  MoveL 4658 to (-31.93, 163.09, 78.65) mm, rotated rx 180 ry 0 rz -180 deg; joints [-126.273, -59.59, -78.383, 61.404, 66.666, -36.002]
  Call Extruder(2.36471)
  MoveL 4659 to (-32.22, 162.97, 78.65) mm, rotated rx 180 ry 0 rz 180 deg; joints [-126.252, -59.57, -78.436, 61.41, 66.694, -35.978]
  MoveL 4660 to (-32.22, 162.97, 78.65) mm, rotated rx 180 ry 0 rz 180 deg; joints [-126.252, -59.57, -78.436, 61.41, 66.694, -35.978]
  Call Extruder(2.53513)
  MoveL 4661 to (-32.49, 162.85, 78.65) mm, rotated rx -180 ry 0 rz -180 deg; joints [-126.233, -59.55, -78.486, 61.416, 66.72, -35.956]
  MoveL 4662 to (-32.49, 162.85, 78.65) mm, rotated rx -180 ry 0 rz -180 deg; joints [-126.233, -59.55, -78.486, 61.416, 66.72, -35.956]
  Call Extruder(2.69310)
  MoveL 4663 to (-32.74, 162.74, 78.65) mm, rotated rx -180 ry 0 rz 180 deg; joints [-126.215, -59.532, -78.531, 61.421, 66.744, -35.936]
  MoveL 4664 to (-32.74, 162.74, 78.65) mm, rotated rx -180 ry 0 rz 180 deg; joints [-126.215, -59.532, -78.531, 61.421, 66.744, -35.936]
  Call Extruder(2.85168)
  MoveL 4665 to (-32.99, 162.64, 78.65) mm, rotated rx 180 ry 0 rz 180 deg; joints [-126.197, -59.514, -78.577, 61.426, 66.767, -35.916]
  MoveL 4666 to (-32.99, 162.64, 78.65) mm, rotated rx 180 ry 0 rz 180 deg; joints [-126.197, -59.514, -78.577, 61.426, 66.767, -35.916]
  Call Extruder(3.05784)
  MoveL 4667 to (-33.29, 162.46, 78.65) mm, rotated rx 180 ry 0 rz -180 deg; joints [-126.179, -59.489, -78.64, 61.428, 66.797, -35.885]
  MoveL 4668 to (-33.29, 162.46, 78.65) mm, rotated rx 180 ry 0 rz -180 deg; joints [-126.179, -59.489, -78.64, 61.428, 66.797, -35.885]
  Call Extruder(3.26479)
  MoveL 4669 to (-33.6, 162.29, 78.65) mm, rotated rx 180 ry 0 rz -180 deg; joints [-126.16, -59.465, -78.703, 61.43, 66.826, -35.855]
  MoveL 4670 to (-33.6, 162.29, 78.65) mm, rotated rx 180 ry 0 rz -180 deg; joints [-126.16, -59.465, -78.703, 61.43, 66.826, -35.855]
  Call Extruder(3.47251)
  MoveL 4671 to (-33.9, 162.11, 78.65) mm, rotated rx 180 ry 0 rz 180 deg; joints [-126.142, -59.44, -78.766, 61.432, 66.855, -35.825]
  MoveL 4672 to (-33.9, 162.11, 78.65) mm, rotated rx 180 ry 0 rz 180 deg; joints [-126.142, -59.44, -78.766, 61.432, 66.855, -35.825]
  Call Extruder(3.68102)
  MoveL 4673 to (-34.21, 161.93, 78.65) mm, rotated rx -180 ry 0 rz 180 deg; joints [-126.123, -59.415, -78.829, 61.434, 66.884, -35.795]
  MoveL 4674 to (-34.21, 161.93, 78.65) mm, rotated rx -180 ry 0 rz 180 deg; joints [-126.123, -59.415, -78.829, 61.434, 66.884, -35.795]
  Call Extruder(3.86055)
  MoveL 4675 to (-34.45, 161.76, 78.65) mm, rotated rx -180 ry 0 rz 180 deg; joints [-126.111, -59.393, -78.885, 61.432, 66.907, -35.767]
  MoveL 4676 to (-34.45, 161.76, 78.65) mm, rotated rx -180 ry 0 rz 180 deg; joints [-126.111, -59.393, -78.885, 61.432, 66.907, -35.767]
  Call Extruder(4.19399)
  MoveL 4677 to (-34.9, 161.43, 78.65) mm, rotated rx 180 ry 0 rz 180 deg; joints [-126.089, -59.353, -78.988, 61.428, 66.95, -35.714]
  MoveL 4678 to (-34.9, 161.43, 78.65) mm, rotated rx 180 ry 0 rz 180 deg; joints [-126.089, -59.353, -78.988, 61.428, 66.95, -35.714]
  Call Extruder(4.52861)
  MoveL 4679 to (-35.35, 161.1, 78.65) mm, rotated rx 180 ry 0 rz -180 deg; joints [-126.067, -59.312, -79.092, 61.424, 66.993, -35.662]
  Call Extruder(5.35652)
  MoveL 4680 to (-36.39, 160.19, 78.65) mm, rotated rx -180 ry 0 rz 180 deg; joints [-126.027, -59.21, -79.355, 61.399, 67.093, -35.523]
  Call Extruder(6.18445)
  MoveL 4681 to (-37.3, 159.15, 78.65) mm, rotated rx -180 ry 0 rz 180 deg; joints [-126.011, -59.106, -79.622, 61.354, 67.181, -35.373]
  Call Extruder(6.35176)
  MoveL 4682 to (-37.47, 158.93, 78.65) mm, rotated rx 180 ry 0 rz 180 deg; joints [-126.011, -59.084, -79.676, 61.341, 67.197, -35.341]
  MoveL 4683 to (-37.47, 158.93, 78.65) mm, rotated rx 180 ry 0 rz 180 deg; joints [-126.011, -59.084, -79.676, 61.341, 67.197, -35.341]
  Call Extruder(6.68519)
  MoveL 4684 to (-37.79, 158.48, 78.65) mm, rotated rx 180 ry 0 rz -180 deg; joints [-126.011, -59.042, -79.784, 61.317, 67.228, -35.279]
  MoveL 4685 to (-37.79, 158.48, 78.65) mm, rotated rx 180 ry 0 rz -180 deg; joints [-126.011, -59.042, -79.784, 61.317, 67.228, -35.279]
  Call Extruder(7.01743)
  MoveL 4686 to (-38.12, 158.02, 78.65) mm, rotated rx 180 ry 0 rz -180 deg; joints [-126.011, -59, -79.893, 61.293, 67.26, -35.216]
  MoveL 4687 to (-38.12, 158.02, 78.65) mm, rotated rx 180 ry 0 rz -180 deg; joints [-126.011, -59, -79.893, 61.293, 67.26, -35.216]
  Call Extruder(7.13511)
  MoveL 4688 to (-38.22, 157.85, 78.65) mm, rotated rx 180 ry 0 rz 180 deg; joints [-126.013, -58.986, -79.931, 61.282, 67.27, -35.192]
  MoveL 4689 to (-38.22, 157.85, 78.65) mm, rotated rx 180 ry 0 rz 180 deg; joints [-126.013, -58.986, -79.931, 61.282, 67.27, -35.192]
  Call Extruder(7.34283)
  MoveL 4690 to (-38.4, 157.55, 78.65) mm, rotated rx 180 ry 0 rz -180 deg; joints [-126.018, -58.959, -79.998, 61.262, 67.287, -35.151]
  MoveL 4691 to (-38.4, 157.55, 78.65) mm, rotated rx 180 ry 0 rz -180 deg; joints [-126.018, -58.959, -79.998, 61.262, 67.287, -35.151]
  Call Extruder(7.54978)
  MoveL 4692 to (-38.57, 157.25, 78.65) mm, rotated rx 180 ry 0 rz 180 deg; joints [-126.023, -58.933, -80.066, 61.243, 67.304, -35.111]
  MoveL 4693 to (-38.57, 157.25, 78.65) mm, rotated rx 180 ry 0 rz 180 deg; joints [-126.023, -58.933, -80.066, 61.243, 67.304, -35.111]
  Call Extruder(7.75595)
  MoveL 4694 to (-38.75, 156.94, 78.65) mm, rotated rx -180 ry 0 rz 180 deg; joints [-126.028, -58.907, -80.133, 61.223, 67.321, -35.07]
  MoveL 4695 to (-38.75, 156.94, 78.65) mm, rotated rx -180 ry 0 rz 180 deg; joints [-126.028, -58.907, -80.133, 61.223, 67.321, -35.07]
  Call Extruder(7.93762)
  MoveL 4696 to (-38.89, 156.66, 78.65) mm, rotated rx 180 ry 0 rz 180 deg; joints [-126.034, -58.884, -80.193, 61.204, 67.335, -35.033]
  MoveL 4697 to (-38.89, 156.66, 78.65) mm, rotated rx 180 ry 0 rz 180 deg; joints [-126.034, -58.884, -80.193, 61.204, 67.335, -35.033]
  Call Extruder(8.09561)
  MoveL 4698 to (-39, 156.42, 78.65) mm, rotated rx 180 ry 0 rz -180 deg; joints [-126.042, -58.864, -80.244, 61.186, 67.345, -35]
  MoveL 4699 to (-39, 156.42, 78.65) mm, rotated rx 180 ry 0 rz -180 deg; joints [-126.042, -58.864, -80.244, 61.186, 67.345, -35]
  Call Extruder(8.25300)
  MoveL 4700 to (-39.1, 156.17, 78.65) mm, rotated rx 180 ry 0 rz 180 deg; joints [-126.05, -58.845, -80.295, 61.167, 67.356, -34.968]
  MoveL 4701 to (-39.1, 156.17, 78.65) mm, rotated rx 180 ry 0 rz 180 deg; joints [-126.05, -58.845, -80.295, 61.167, 67.356, -34.968]
  Call Extruder(8.43572)
  MoveL 4702 to (-39.23, 155.88, 78.65) mm, rotated rx 180 ry 0 rz 180 deg; joints [-126.06, -58.822, -80.354, 61.145, 67.368, -34.93]
  MoveL 4703 to (-39.23, 155.88, 78.65) mm, rotated rx 180 ry 0 rz 180 deg; joints [-126.06, -58.822, -80.354, 61.145, 67.368, -34.93]
  Call Extruder(8.61768)
  MoveL 4704 to (-39.35, 155.58, 78.65) mm, rotated rx -180 ry 0 rz -180 deg; joints [-126.07, -58.799, -80.413, 61.123, 67.38, -34.892]
  MoveL 4705 to (-39.35, 155.58, 78.65) mm, rotated rx -180 ry 0 rz -180 deg; joints [-126.07, -58.799, -80.413, 61.123, 67.38, -34.892]
  Call Extruder(8.76501)
  MoveL 4706 to (-39.44, 155.34, 78.65) mm, rotated rx 180 ry 0 rz 180 deg; joints [-126.079, -58.78, -80.461, 61.105, 67.389, -34.862]
  MoveL 4707 to (-39.44, 155.34, 78.65) mm, rotated rx 180 ry 0 rz 180 deg; joints [-126.079, -58.78, -80.461, 61.105, 67.389, -34.862]
  Call Extruder(8.87825)
  MoveL 4708 to (-39.5, 155.15, 78.65) mm, rotated rx -180 ry 0 rz 180 deg; joints [-126.087, -58.766, -80.497, 61.089, 67.395, -34.838]
  MoveL 4709 to (-39.5, 155.15, 78.65) mm, rotated rx -180 ry 0 rz 180 deg; joints [-126.087, -58.766, -80.497, 61.089, 67.395, -34.838]
  Call Extruder(8.99103)
  MoveL 4710 to (-39.56, 154.97, 78.65) mm, rotated rx 180 ry 0 rz 180 deg; joints [-126.095, -58.752, -80.533, 61.074, 67.401, -34.814]
  MoveL 4711 to (-39.56, 154.97, 78.65) mm, rotated rx 180 ry 0 rz 180 deg; joints [-126.095, -58.752, -80.533, 61.074, 67.401, -34.814]
  Call Extruder(9.10338)
  MoveL 4712 to (-39.62, 154.78, 78.65) mm, rotated rx 180 ry 0 rz 180 deg; joints [-126.103, -58.738, -80.57, 61.059, 67.407, -34.79]
  MoveL 4713 to (-39.62, 154.78, 78.65) mm, rotated rx 180 ry 0 rz 180 deg; joints [-126.103, -58.738, -80.57, 61.059, 67.407, -34.79]
  Call Extruder(9.21528)
  MoveL 4714 to (-39.68, 154.59, 78.65) mm, rotated rx -180 ry 0 rz 180 deg; joints [-126.111, -58.725, -80.606, 61.043, 67.413, -34.766]
  MoveL 4715 to (-39.68, 154.59, 78.65) mm, rotated rx -180 ry 0 rz 180 deg; joints [-126.111, -58.725, -80.606, 61.043, 67.413, -34.766]
  Call Extruder(9.33668)
  MoveL 4716 to (-39.75, 154.38, 78.65) mm, rotated rx -180 ry 0 rz 180 deg; joints [-126.12, -58.709, -80.645, 61.026, 67.42, -34.74]
  MoveL 4717 to (-39.75, 154.38, 78.65) mm, rotated rx -180 ry 0 rz 180 deg; joints [-126.12, -58.709, -80.645, 61.026, 67.42, -34.74]
  Call Extruder(9.46748)
  MoveL 4718 to (-39.81, 154.16, 78.65) mm, rotated rx 180 ry 0 rz 180 deg; joints [-126.131, -58.693, -80.688, 61.008, 67.427, -34.712]
  MoveL 4719 to (-39.81, 154.16, 78.65) mm, rotated rx 180 ry 0 rz 180 deg; joints [-126.131, -58.693, -80.688, 61.008, 67.427, -34.712]
  Call Extruder(9.59770)
  MoveL 4720 to (-39.88, 153.94, 78.65) mm, rotated rx 180 ry 0 rz 180 deg; joints [-126.141, -58.677, -80.73, 60.989, 67.433, -34.684]
  MoveL 4721 to (-39.88, 153.94, 78.65) mm, rotated rx 180 ry 0 rz 180 deg; joints [-126.141, -58.677, -80.73, 60.989, 67.433, -34.684]
  Call Extruder(9.72737)
  MoveL 4722 to (-39.95, 153.71, 78.65) mm, rotated rx 180 ry 0 rz 180 deg; joints [-126.151, -58.66, -80.772, 60.971, 67.44, -34.655]
  MoveL 4723 to (-39.95, 153.71, 78.65) mm, rotated rx 180 ry 0 rz 180 deg; joints [-126.151, -58.66, -80.772, 60.971, 67.44, -34.655]
  Call Extruder(9.85647)
  MoveL 4724 to (-40.02, 153.49, 78.65) mm, rotated rx -180 ry 0 rz -180 deg; joints [-126.161, -58.644, -80.815, 60.952, 67.447, -34.627]
  MoveL 4725 to (-40.02, 153.49, 78.65) mm, rotated rx -180 ry 0 rz -180 deg; joints [-126.161, -58.644, -80.815, 60.952, 67.447, -34.627]
  Call Extruder(9.97156)
  MoveL 4726 to (-40.06, 153.28, 78.65) mm, rotated rx -180 ry 0 rz 180 deg; joints [-126.173, -58.63, -80.851, 60.934, 67.452, -34.602]
  MoveL 4727 to (-40.06, 153.28, 78.65) mm, rotated rx -180 ry 0 rz 180 deg; joints [-126.173, -58.63, -80.851, 60.934, 67.452, -34.602]
  Call Extruder(10.08619)
  MoveL 4728 to (-40.11, 153.08, 78.65) mm, rotated rx 180 ry 0 rz -180 deg; joints [-126.184, -58.616, -80.888, 60.916, 67.456, -34.577]
  MoveL 4729 to (-40.11, 153.08, 78.65) mm, rotated rx 180 ry 0 rz -180 deg; joints [-126.184, -58.616, -80.888, 60.916, 67.456, -34.577]
  Call Extruder(10.20037)
  MoveL 4730 to (-40.15, 152.88, 78.65) mm, rotated rx 180 ry 0 rz 180 deg; joints [-126.195, -58.602, -80.925, 60.897, 67.461, -34.552]
  MoveL 4731 to (-40.15, 152.88, 78.65) mm, rotated rx 180 ry 0 rz 180 deg; joints [-126.195, -58.602, -80.925, 60.897, 67.461, -34.552]
  Call Extruder(10.31410)
  MoveL 4732 to (-40.2, 152.67, 78.65) mm, rotated rx 180 ry 0 rz 180 deg; joints [-126.206, -58.588, -80.961, 60.879, 67.465, -34.526]
  MoveL 4733 to (-40.2, 152.67, 78.65) mm, rotated rx 180 ry 0 rz 180 deg; joints [-126.206, -58.588, -80.961, 60.879, 67.465, -34.526]
  Call Extruder(10.43953)
  MoveL 4734 to (-40.24, 152.44, 78.65) mm, rotated rx 180 ry 0 rz 180 deg; joints [-126.219, -58.572, -81.002, 60.859, 67.47, -34.499]
  MoveL 4735 to (-40.24, 152.44, 78.65) mm, rotated rx 180 ry 0 rz 180 deg; joints [-126.219, -58.572, -81.002, 60.859, 67.47, -34.499]
  Call Extruder(10.57650)
  MoveL 4736 to (-40.29, 152.2, 78.65) mm, rotated rx 180 ry 0 rz -180 deg; joints [-126.233, -58.555, -81.046, 60.836, 67.476, -34.468]
  MoveL 4737 to (-40.29, 152.2, 78.65) mm, rotated rx 180 ry 0 rz -180 deg; joints [-126.233, -58.555, -81.046, 60.836, 67.476, -34.468]
  Call Extruder(10.71287)
  MoveL 4738 to (-40.34, 151.95, 78.65) mm, rotated rx 180 ry 0 rz 180 deg; joints [-126.248, -58.538, -81.09, 60.814, 67.481, -34.437]
  MoveL 4739 to (-40.34, 151.95, 78.65) mm, rotated rx 180 ry 0 rz 180 deg; joints [-126.248, -58.538, -81.09, 60.814, 67.481, -34.437]
  Call Extruder(10.84862)
  MoveL 4740 to (-40.39, 151.7, 78.65) mm, rotated rx 180 ry 0 rz 180 deg; joints [-126.262, -58.521, -81.134, 60.791, 67.486, -34.407]
  MoveL 4741 to (-40.39, 151.7, 78.65) mm, rotated rx 180 ry 0 rz 180 deg; joints [-126.262, -58.521, -81.134, 60.791, 67.486, -34.407]
  Call Extruder(10.98377)
  MoveL 4742 to (-40.44, 151.45, 78.65) mm, rotated rx 180 ry 0 rz 180 deg; joints [-126.276, -58.505, -81.178, 60.768, 67.491, -34.376]
  MoveL 4743 to (-40.44, 151.45, 78.65) mm, rotated rx 180 ry 0 rz 180 deg; joints [-126.276, -58.505, -81.178, 60.768, 67.491, -34.376]
  Call Extruder(11.11830)
  MoveL 4744 to (-40.49, 151.2, 78.65) mm, rotated rx 180 ry 0 rz 180 deg; joints [-126.291, -58.488, -81.222, 60.746, 67.496, -34.346]
  MoveL 4745 to (-40.49, 151.2, 78.65) mm, rotated rx 180 ry 0 rz 180 deg; joints [-126.291, -58.488, -81.222, 60.746, 67.496, -34.346]
  Call Extruder(11.25223)
  MoveL 4746 to (-40.54, 150.95, 78.65) mm, rotated rx -180 ry 0 rz 180 deg; joints [-126.305, -58.471, -81.266, 60.723, 67.501, -34.315]
  MoveL 4747 to (-40.54, 150.95, 78.65) mm, rotated rx -180 ry 0 rz 180 deg; joints [-126.305, -58.471, -81.266, 60.723, 67.501, -34.315]
  Call Extruder(11.40008)
  MoveL 4748 to (-40.59, 150.67, 78.65) mm, rotated rx -180 ry 0 rz 180 deg; joints [-126.322, -58.452, -81.314, 60.697, 67.506, -34.281]
  MoveL 4749 to (-40.59, 150.67, 78.65) mm, rotated rx -180 ry 0 rz 180 deg; joints [-126.322, -58.452, -81.314, 60.697, 67.506, -34.281]
  Call Extruder(11.56181)
  MoveL 4750 to (-40.64, 150.37, 78.65) mm, rotated rx -180 ry 0 rz -180 deg; joints [-126.341, -58.432, -81.367, 60.669, 67.512, -34.244]
  MoveL 4751 to (-40.64, 150.37, 78.65) mm, rotated rx -180 ry 0 rz -180 deg; joints [-126.341, -58.432, -81.367, 60.669, 67.512, -34.244]
  Call Extruder(11.72281)
  MoveL 4752 to (-40.69, 150.06, 78.65) mm, rotated rx 180 ry 0 rz -180 deg; joints [-126.36, -58.412, -81.419, 60.64, 67.517, -34.207]
  MoveL 4753 to (-40.69, 150.06, 78.65) mm, rotated rx 180 ry 0 rz -180 deg; joints [-126.36, -58.412, -81.419, 60.64, 67.517, -34.207]
  Call Extruder(11.88308)
  MoveL 4754 to (-40.74, 149.76, 78.65) mm, rotated rx -180 ry 0 rz 180 deg; joints [-126.379, -58.392, -81.472, 60.611, 67.522, -34.17]
  MoveL 4755 to (-40.74, 149.76, 78.65) mm, rotated rx -180 ry 0 rz 180 deg; joints [-126.379, -58.392, -81.472, 60.611, 67.522, -34.17]
  Call Extruder(12.04262)
  MoveL 4756 to (-40.78, 149.45, 78.65) mm, rotated rx 180 ry 0 rz 180 deg; joints [-126.398, -58.372, -81.524, 60.583, 67.527, -34.133]
  MoveL 4757 to (-40.78, 149.45, 78.65) mm, rotated rx 180 ry 0 rz 180 deg; joints [-126.398, -58.372, -81.524, 60.583, 67.527, -34.133]
  Call Extruder(12.20143)
  MoveL 4758 to (-40.83, 149.14, 78.65) mm, rotated rx -180 ry 0 rz 180 deg; joints [-126.417, -58.352, -81.577, 60.554, 67.533, -34.096]
  MoveL 4759 to (-40.83, 149.14, 78.65) mm, rotated rx -180 ry 0 rz 180 deg; joints [-126.417, -58.352, -81.577, 60.554, 67.533, -34.096]
  Call Extruder(12.38010)
  MoveL 4760 to (-40.88, 148.8, 78.65) mm, rotated rx -180 ry 0 rz 180 deg; joints [-126.439, -58.33, -81.635, 60.521, 67.538, -34.054]
  MoveL 4761 to (-40.88, 148.8, 78.65) mm, rotated rx -180 ry 0 rz 180 deg; joints [-126.439, -58.33, -81.635, 60.521, 67.538, -34.054]
  Call Extruder(12.57854)
  MoveL 4762 to (-40.92, 148.41, 78.65) mm, rotated rx 180 ry 0 rz -180 deg; joints [-126.465, -58.305, -81.7, 60.483, 67.543, -34.008]
  MoveL 4763 to (-40.92, 148.41, 78.65) mm, rotated rx 180 ry 0 rz -180 deg; joints [-126.465, -58.305, -81.7, 60.483, 67.543, -34.008]
  Call Extruder(12.77611)
  MoveL 4764 to (-40.97, 148.02, 78.65) mm, rotated rx 180 ry 0 rz -180 deg; joints [-126.491, -58.281, -81.764, 60.445, 67.548, -33.961]
  MoveL 4765 to (-40.97, 148.02, 78.65) mm, rotated rx 180 ry 0 rz -180 deg; joints [-126.491, -58.281, -81.764, 60.445, 67.548, -33.961]
  Call Extruder(12.97282)
  MoveL 4766 to (-41.02, 147.63, 78.65) mm, rotated rx 180 ry 0 rz 180 deg; joints [-126.517, -58.256, -81.829, 60.408, 67.553, -33.915]
  MoveL 4767 to (-41.02, 147.63, 78.65) mm, rotated rx 180 ry 0 rz 180 deg; joints [-126.517, -58.256, -81.829, 60.408, 67.553, -33.915]
  Call Extruder(13.16866)
  MoveL 4768 to (-41.06, 147.25, 78.65) mm, rotated rx -180 ry 0 rz -180 deg; joints [-126.543, -58.232, -81.893, 60.37, 67.558, -33.868]
  MoveL 4769 to (-41.06, 147.25, 78.65) mm, rotated rx -180 ry 0 rz -180 deg; joints [-126.543, -58.232, -81.893, 60.37, 67.558, -33.868]
  Call Extruder(13.46406)
  MoveL 4770 to (-41.11, 146.66, 78.65) mm, rotated rx -180 ry 0 rz -180 deg; joints [-126.585, -58.195, -81.988, 60.311, 67.564, -33.798]
  MoveL 4771 to (-41.11, 146.66, 78.65) mm, rotated rx -180 ry 0 rz -180 deg; joints [-126.585, -58.195, -81.988, 60.311, 67.564, -33.798]
  Call Extruder(13.75812)
  MoveL 4772 to (-41.15, 146.07, 78.65) mm, rotated rx -180 ry 0 rz -180 deg; joints [-126.628, -58.159, -82.083, 60.252, 67.57, -33.728]
  MoveL 4773 to (-41.15, 146.07, 78.65) mm, rotated rx -180 ry 0 rz -180 deg; joints [-126.628, -58.159, -82.083, 60.252, 67.57, -33.728]
  Call Extruder(14.05086)
  MoveL 4774 to (-41.2, 145.48, 78.65) mm, rotated rx 180 ry 0 rz 180 deg; joints [-126.67, -58.123, -82.178, 60.192, 67.576, -33.658]
  MoveL 4775 to (-41.2, 145.48, 78.65) mm, rotated rx 180 ry 0 rz 180 deg; joints [-126.67, -58.123, -82.178, 60.192, 67.576, -33.658]
  Call Extruder(14.62431)
  MoveL 4776 to (-41.25, 144.32, 78.65) mm, rotated rx 180 ry 0 rz 180 deg; joints [-126.759, -58.054, -82.36, 60.072, 67.583, -33.522]
  MoveL 4777 to (-41.25, 144.32, 78.65) mm, rotated rx 180 ry 0 rz 180 deg; joints [-126.759, -58.054, -82.36, 60.072, 67.583, -33.522]
  Call Extruder(15.33827)
  MoveL 4778 to (-41.29, 142.86, 78.65) mm, rotated rx 180 ry 0 rz -180 deg; joints [-126.873, -57.969, -82.585, 59.919, 67.59, -33.352]
  Call Extruder(57.40309)
  MoveL 4779 to (-41.29, 57.14, 78.65) mm, rotated rx 180 ry 0 rz 180 deg; joints [-135.148, -53.894, -94.222, 49.519, 68.009, -23.688]
  Call Extruder(57.83164)
  MoveL 4780 to (-41.27, 56.26, 78.65) mm, rotated rx -180 ry 0 rz -180 deg; joints [-135.25, -53.862, -94.325, 49.397, 68.014, -23.593]
  MoveL 4781 to (-41.27, 56.26, 78.65) mm, rotated rx -180 ry 0 rz -180 deg; joints [-135.25, -53.862, -94.325, 49.397, 68.014, -23.593]
  Call Extruder(58.40509)
  MoveL 4782 to (-41.22, 55.1, 78.65) mm, rotated rx 180 ry 0 rz 180 deg; joints [-135.387, -53.819, -94.459, 49.232, 68.019, -23.467]
  MoveL 4783 to (-41.22, 55.1, 78.65) mm, rotated rx 180 ry 0 rz 180 deg; joints [-135.387, -53.819, -94.459, 49.232, 68.019, -23.467]
  Call Extruder(58.83941)
  MoveL 4784 to (-41.18, 54.23, 78.65) mm, rotated rx 180 ry 0 rz 180 deg; joints [-135.493, -53.788, -94.558, 49.107, 68.021, -23.372]
  MoveL 4785 to (-41.18, 54.23, 78.65) mm, rotated rx 180 ry 0 rz 180 deg; joints [-135.493, -53.788, -94.558, 49.107, 68.021, -23.372]
  Call Extruder(59.13347)
  MoveL 4786 to (-41.13, 53.64, 78.65) mm, rotated rx -180 ry 0 rz 180 deg; joints [-135.566, -53.767, -94.623, 49.021, 68.021, -23.309]
  MoveL 4787 to (-41.13, 53.64, 78.65) mm, rotated rx -180 ry 0 rz 180 deg; joints [-135.566, -53.767, -94.623, 49.021, 68.021, -23.309]
  Call Extruder(59.42887)
  MoveL 4788 to (-41.09, 53.05, 78.65) mm, rotated rx 180 ry 0 rz 180 deg; joints [-135.64, -53.747, -94.687, 48.935, 68.021, -23.246]
  MoveL 4789 to (-41.09, 53.05, 78.65) mm, rotated rx 180 ry 0 rz 180 deg; joints [-135.64, -53.747, -94.687, 48.935, 68.021, -23.246]
  Call Extruder(59.67511)
  MoveL 4790 to (-41.04, 52.56, 78.65) mm, rotated rx 180 ry 0 rz 180 deg; joints [-135.701, -53.731, -94.74, 48.863, 68.021, -23.194]
  MoveL 4791 to (-41.04, 52.56, 78.65) mm, rotated rx 180 ry 0 rz 180 deg; joints [-135.701, -53.731, -94.74, 48.863, 68.021, -23.194]
  Call Extruder(59.87182)
  MoveL 4792 to (-40.99, 52.17, 78.65) mm, rotated rx 180 ry 0 rz 180 deg; joints [-135.751, -53.718, -94.78, 48.805, 68.019, -23.153]
  MoveL 4793 to (-40.99, 52.17, 78.65) mm, rotated rx 180 ry 0 rz 180 deg; joints [-135.751, -53.718, -94.78, 48.805, 68.019, -23.153]
  Call Extruder(60.06939)
  MoveL 4794 to (-40.95, 51.78, 78.65) mm, rotated rx -180 ry 0 rz -180 deg; joints [-135.801, -53.705, -94.82, 48.747, 68.018, -23.112]
  MoveL 4795 to (-40.95, 51.78, 78.65) mm, rotated rx -180 ry 0 rz -180 deg; joints [-135.801, -53.705, -94.82, 48.747, 68.018, -23.112]
  Call Extruder(60.26783)
  MoveL 4796 to (-40.9, 51.4, 78.65) mm, rotated rx 180 ry 0 rz -180 deg; joints [-135.852, -53.692, -94.861, 48.689, 68.016, -23.071]
  MoveL 4797 to (-40.9, 51.4, 78.65) mm, rotated rx 180 ry 0 rz -180 deg; joints [-135.852, -53.692, -94.861, 48.689, 68.016, -23.071]
  Call Extruder(60.46714)
  MoveL 4798 to (-40.86, 51.01, 78.65) mm, rotated rx -180 ry 0 rz 180 deg; joints [-135.902, -53.68, -94.901, 48.63, 68.015, -23.03]
  MoveL 4799 to (-40.86, 51.01, 78.65) mm, rotated rx -180 ry 0 rz 180 deg; joints [-135.902, -53.68, -94.901, 48.63, 68.015, -23.03]
  Call Extruder(60.62596)
  MoveL 4800 to (-40.81, 50.7, 78.65) mm, rotated rx 180 ry 0 rz -180 deg; joints [-135.943, -53.67, -94.931, 48.583, 68.012, -22.998]
  MoveL 4801 to (-40.81, 50.7, 78.65) mm, rotated rx 180 ry 0 rz -180 deg; joints [-135.943, -53.67, -94.931, 48.583, 68.012, -22.998]
  Call Extruder(60.78550)
  MoveL 4802 to (-40.76, 50.4, 78.65) mm, rotated rx 180 ry 0 rz -180 deg; joints [-135.984, -53.661, -94.961, 48.536, 68.01, -22.966]
  MoveL 4803 to (-40.76, 50.4, 78.65) mm, rotated rx 180 ry 0 rz -180 deg; joints [-135.984, -53.661, -94.961, 48.536, 68.01, -22.966]
  Call Extruder(60.94577)
  MoveL 4804 to (-40.71, 50.09, 78.65) mm, rotated rx 180 ry 0 rz 180 deg; joints [-136.025, -53.652, -94.992, 48.489, 68.008, -22.934]
  MoveL 4805 to (-40.71, 50.09, 78.65) mm, rotated rx 180 ry 0 rz 180 deg; joints [-136.025, -53.652, -94.992, 48.489, 68.008, -22.934]
  Call Extruder(61.10677)
  MoveL 4806 to (-40.66, 49.79, 78.65) mm, rotated rx 180 ry 0 rz -180 deg; joints [-136.067, -53.642, -95.022, 48.442, 68.005, -22.902]
  MoveL 4807 to (-40.66, 49.79, 78.65) mm, rotated rx 180 ry 0 rz -180 deg; joints [-136.067, -53.642, -95.022, 48.442, 68.005, -22.902]
  Call Extruder(61.26850)
  MoveL 4808 to (-40.61, 49.48, 78.65) mm, rotated rx 180 ry 0 rz 180 deg; joints [-136.108, -53.633, -95.052, 48.395, 68.003, -22.87]
  MoveL 4809 to (-40.61, 49.48, 78.65) mm, rotated rx 180 ry 0 rz 180 deg; joints [-136.108, -53.633, -95.052, 48.395, 68.003, -22.87]
  Call Extruder(61.43095)
  MoveL 4810 to (-40.56, 49.18, 78.65) mm, rotated rx 180 ry 0 rz 180 deg; joints [-136.149, -53.623, -95.082, 48.347, 68.001, -22.838]
  MoveL 4811 to (-40.56, 49.18, 78.65) mm, rotated rx 180 ry 0 rz 180 deg; joints [-136.149, -53.623, -95.082, 48.347, 68.001, -22.838]
  Call Extruder(61.56487)
  MoveL 4812 to (-40.52, 48.92, 78.65) mm, rotated rx -180 ry 0 rz 180 deg; joints [-136.184, -53.616, -95.105, 48.308, 67.998, -22.812]
  MoveL 4813 to (-40.52, 48.92, 78.65) mm, rotated rx -180 ry 0 rz 180 deg; joints [-136.184, -53.616, -95.105, 48.308, 67.998, -22.812]
  Call Extruder(61.69941)
  MoveL 4814 to (-40.47, 48.68, 78.65) mm, rotated rx -180 ry 0 rz 180 deg; joints [-136.219, -53.609, -95.128, 48.269, 67.995, -22.786]
  MoveL 4815 to (-40.47, 48.68, 78.65) mm, rotated rx -180 ry 0 rz 180 deg; joints [-136.219, -53.609, -95.128, 48.269, 67.995, -22.786]
  Call Extruder(61.83455)
  MoveL 4816 to (-40.42, 48.43, 78.65) mm, rotated rx 180 ry 0 rz 180 deg; joints [-136.254, -53.602, -95.151, 48.229, 67.992, -22.76]
  MoveL 4817 to (-40.42, 48.43, 78.65) mm, rotated rx 180 ry 0 rz 180 deg; joints [-136.254, -53.602, -95.151, 48.229, 67.992, -22.76]
  Call Extruder(61.97031)
  MoveL 4818 to (-40.37, 48.18, 78.65) mm, rotated rx 180 ry 0 rz 180 deg; joints [-136.288, -53.594, -95.174, 48.19, 67.989, -22.734]
  MoveL 4819 to (-40.37, 48.18, 78.65) mm, rotated rx 180 ry 0 rz 180 deg; joints [-136.288, -53.594, -95.174, 48.19, 67.989, -22.734]
  Call Extruder(62.10667)
  MoveL 4820 to (-40.32, 47.93, 78.65) mm, rotated rx -180 ry 0 rz 180 deg; joints [-136.323, -53.587, -95.197, 48.15, 67.986, -22.709]
  MoveL 4821 to (-40.32, 47.93, 78.65) mm, rotated rx -180 ry 0 rz 180 deg; joints [-136.323, -53.587, -95.197, 48.15, 67.986, -22.709]
  Call Extruder(62.24365)
  MoveL 4822 to (-40.27, 47.68, 78.65) mm, rotated rx 180 ry 0 rz 180 deg; joints [-136.358, -53.58, -95.221, 48.111, 67.983, -22.683]
  MoveL 4823 to (-40.27, 47.68, 78.65) mm, rotated rx 180 ry 0 rz 180 deg; joints [-136.358, -53.58, -95.221, 48.111, 67.983, -22.683]
  Call Extruder(62.38124)
  MoveL 4824 to (-40.22, 47.43, 78.65) mm, rotated rx 180 ry 0 rz 180 deg; joints [-136.393, -53.573, -95.243, 48.071, 67.981, -22.657]
  MoveL 4825 to (-40.22, 47.43, 78.65) mm, rotated rx 180 ry 0 rz 180 deg; joints [-136.393, -53.573, -95.243, 48.071, 67.981, -22.657]
  Call Extruder(62.49496)
  MoveL 4826 to (-40.17, 47.23, 78.65) mm, rotated rx 180 ry 0 rz -180 deg; joints [-136.422, -53.567, -95.262, 48.038, 67.978, -22.636]
  MoveL 4827 to (-40.17, 47.23, 78.65) mm, rotated rx 180 ry 0 rz -180 deg; joints [-136.422, -53.567, -95.262, 48.038, 67.978, -22.636]
  Call Extruder(62.60914)
  MoveL 4828 to (-40.13, 47.02, 78.65) mm, rotated rx 180 ry 0 rz 180 deg; joints [-136.452, -53.561, -95.28, 48.005, 67.975, -22.615]
  MoveL 4829 to (-40.13, 47.02, 78.65) mm, rotated rx 180 ry 0 rz 180 deg; joints [-136.452, -53.561, -95.28, 48.005, 67.975, -22.615]
  Call Extruder(62.72378)
  MoveL 4830 to (-40.08, 46.82, 78.65) mm, rotated rx 180 ry 0 rz 180 deg; joints [-136.481, -53.556, -95.299, 47.972, 67.972, -22.594]
  MoveL 4831 to (-40.08, 46.82, 78.65) mm, rotated rx 180 ry 0 rz 180 deg; joints [-136.481, -53.556, -95.299, 47.972, 67.972, -22.594]
  Call Extruder(62.83886)
  MoveL 4832 to (-40.04, 46.61, 78.65) mm, rotated rx -180 ry 0 rz 180 deg; joints [-136.51, -53.55, -95.317, 47.94, 67.97, -22.573]
  MoveL 4833 to (-40.04, 46.61, 78.65) mm, rotated rx -180 ry 0 rz 180 deg; joints [-136.51, -53.55, -95.317, 47.94, 67.97, -22.573]
  Call Extruder(62.96110)
  MoveL 4834 to (-39.98, 46.4, 78.65) mm, rotated rx 180 ry 0 rz 180 deg; joints [-136.542, -53.544, -95.335, 47.904, 67.966, -22.551]
  MoveL 4835 to (-39.98, 46.4, 78.65) mm, rotated rx 180 ry 0 rz 180 deg; joints [-136.542, -53.544, -95.335, 47.904, 67.966, -22.551]
  Call Extruder(63.09076)
  MoveL 4836 to (-39.92, 46.18, 78.65) mm, rotated rx 180 ry 0 rz 180 deg; joints [-136.576, -53.539, -95.353, 47.867, 67.961, -22.529]
  MoveL 4837 to (-39.92, 46.18, 78.65) mm, rotated rx 180 ry 0 rz 180 deg; joints [-136.576, -53.539, -95.353, 47.867, 67.961, -22.529]
  Call Extruder(63.22099)
  MoveL 4838 to (-39.85, 45.95, 78.65) mm, rotated rx 180 ry 0 rz 180 deg; joints [-136.61, -53.533, -95.37, 47.829, 67.956, -22.506]
  MoveL 4839 to (-39.85, 45.95, 78.65) mm, rotated rx 180 ry 0 rz 180 deg; joints [-136.61, -53.533, -95.37, 47.829, 67.956, -22.506]
  Call Extruder(63.35179)
  MoveL 4840 to (-39.78, 45.73, 78.65) mm, rotated rx -180 ry 0 rz -180 deg; joints [-136.644, -53.528, -95.388, 47.791, 67.951, -22.484]
  MoveL 4841 to (-39.78, 45.73, 78.65) mm, rotated rx -180 ry 0 rz -180 deg; joints [-136.644, -53.528, -95.388, 47.791, 67.951, -22.484]
  Call Extruder(63.48315)
  MoveL 4842 to (-39.71, 45.51, 78.65) mm, rotated rx 180 ry 0 rz -180 deg; joints [-136.678, -53.522, -95.406, 47.753, 67.946, -22.461]
  MoveL 4843 to (-39.71, 45.51, 78.65) mm, rotated rx 180 ry 0 rz -180 deg; joints [-136.678, -53.522, -95.406, 47.753, 67.946, -22.461]
  Call Extruder(63.59505)
  MoveL 4844 to (-39.65, 45.32, 78.65) mm, rotated rx -180 ry 0 rz -180 deg; joints [-136.707, -53.518, -95.42, 47.721, 67.942, -22.442]
  MoveL 4845 to (-39.65, 45.32, 78.65) mm, rotated rx -180 ry 0 rz -180 deg; joints [-136.707, -53.518, -95.42, 47.721, 67.942, -22.442]
  Call Extruder(63.70739)
  MoveL 4846 to (-39.59, 45.13, 78.65) mm, rotated rx 180 ry 0 rz 180 deg; joints [-136.737, -53.514, -95.434, 47.689, 67.937, -22.423]
  MoveL 4847 to (-39.59, 45.13, 78.65) mm, rotated rx 180 ry 0 rz 180 deg; joints [-136.737, -53.514, -95.434, 47.689, 67.937, -22.423]
  Call Extruder(63.82018)
  MoveL 4848 to (-39.53, 44.94, 78.65) mm, rotated rx 180 ry 0 rz 180 deg; joints [-136.766, -53.509, -95.449, 47.657, 67.933, -22.405]
  MoveL 4849 to (-39.53, 44.94, 78.65) mm, rotated rx 180 ry 0 rz 180 deg; joints [-136.766, -53.509, -95.449, 47.657, 67.933, -22.405]
  Call Extruder(63.93342)
  MoveL 4850 to (-39.47, 44.75, 78.65) mm, rotated rx 180 ry 0 rz -180 deg; joints [-136.796, -53.505, -95.463, 47.625, 67.928, -22.386]
  MoveL 4851 to (-39.47, 44.75, 78.65) mm, rotated rx 180 ry 0 rz -180 deg; joints [-136.796, -53.505, -95.463, 47.625, 67.928, -22.386]
  Call Extruder(64.04710)
  MoveL 4852 to (-39.41, 44.56, 78.65) mm, rotated rx 180 ry 0 rz 180 deg; joints [-136.825, -53.5, -95.477, 47.592, 67.923, -22.367]
  MoveL 4853 to (-39.41, 44.56, 78.65) mm, rotated rx 180 ry 0 rz 180 deg; joints [-136.825, -53.5, -95.477, 47.592, 67.923, -22.367]
  Call Extruder(64.22906)
  MoveL 4854 to (-39.29, 44.27, 78.65) mm, rotated rx 180 ry 0 rz -180 deg; joints [-136.873, -53.495, -95.496, 47.54, 67.914, -22.338]
  MoveL 4855 to (-39.29, 44.27, 78.65) mm, rotated rx 180 ry 0 rz -180 deg; joints [-136.873, -53.495, -95.496, 47.54, 67.914, -22.338]
  Call Extruder(64.41178)
  MoveL 4856 to (-39.16, 43.98, 78.65) mm, rotated rx 180 ry 0 rz 180 deg; joints [-136.922, -53.489, -95.515, 47.488, 67.904, -22.31]
  MoveL 4857 to (-39.16, 43.98, 78.65) mm, rotated rx 180 ry 0 rz 180 deg; joints [-136.922, -53.489, -95.515, 47.488, 67.904, -22.31]
  Call Extruder(64.58219)
  MoveL 4858 to (-39.05, 43.71, 78.65) mm, rotated rx -180 ry 0 rz 180 deg; joints [-136.967, -53.483, -95.532, 47.439, 67.895, -22.283]
  MoveL 4859 to (-39.05, 43.71, 78.65) mm, rotated rx -180 ry 0 rz 180 deg; joints [-136.967, -53.483, -95.532, 47.439, 67.895, -22.283]
  Call Extruder(64.74017)
  MoveL 4860 to (-38.94, 43.46, 78.65) mm, rotated rx 180 ry 0 rz 180 deg; joints [-137.009, -53.479, -95.547, 47.394, 67.886, -22.259]
  MoveL 4861 to (-38.94, 43.46, 78.65) mm, rotated rx 180 ry 0 rz 180 deg; joints [-137.009, -53.479, -95.547, 47.394, 67.886, -22.259]
  Call Extruder(64.89876)
  MoveL 4862 to (-38.84, 43.21, 78.65) mm, rotated rx -180 ry 0 rz 180 deg; joints [-137.05, -53.474, -95.563, 47.349, 67.878, -22.235]
  MoveL 4863 to (-38.84, 43.21, 78.65) mm, rotated rx -180 ry 0 rz 180 deg; joints [-137.05, -53.474, -95.563, 47.349, 67.878, -22.235]
  Call Extruder(65.10492)
  MoveL 4864 to (-38.66, 42.91, 78.65) mm, rotated rx 180 ry 0 rz -180 deg; joints [-137.107, -53.47, -95.576, 47.291, 67.863, -22.207]
  MoveL 4865 to (-38.66, 42.91, 78.65) mm, rotated rx 180 ry 0 rz -180 deg; joints [-137.107, -53.47, -95.576, 47.291, 67.863, -22.207]
  Call Extruder(65.31187)
  MoveL 4866 to (-38.49, 42.6, 78.65) mm, rotated rx -180 ry 0 rz -180 deg; joints [-137.163, -53.466, -95.589, 47.232, 67.848, -22.178]
  MoveL 4867 to (-38.49, 42.6, 78.65) mm, rotated rx -180 ry 0 rz -180 deg; joints [-137.163, -53.466, -95.589, 47.232, 67.848, -22.178]
  Call Extruder(65.51959)
  MoveL 4868 to (-38.31, 42.3, 78.65) mm, rotated rx 180 ry 0 rz 180 deg; joints [-137.219, -53.462, -95.603, 47.173, 67.833, -22.15]
  MoveL 4869 to (-38.31, 42.3, 78.65) mm, rotated rx 180 ry 0 rz 180 deg; joints [-137.219, -53.462, -95.603, 47.173, 67.833, -22.15]
  Call Extruder(65.72809)
  MoveL 4870 to (-38.13, 41.99, 78.65) mm, rotated rx 180 ry 0 rz 180 deg; joints [-137.275, -53.458, -95.616, 47.114, 67.818, -22.121]
  MoveL 4871 to (-38.13, 41.99, 78.65) mm, rotated rx 180 ry 0 rz 180 deg; joints [-137.275, -53.458, -95.616, 47.114, 67.818, -22.121]
  Call Extruder(65.90765)
  MoveL 4872 to (-37.96, 41.75, 78.65) mm, rotated rx 180 ry 0 rz 180 deg; joints [-137.324, -53.456, -95.622, 47.064, 67.802, -22.099]
  MoveL 4873 to (-37.96, 41.75, 78.65) mm, rotated rx 180 ry 0 rz 180 deg; joints [-137.324, -53.456, -95.622, 47.064, 67.802, -22.099]
  Call Extruder(66.24108)
  MoveL 4874 to (-37.63, 41.3, 78.65) mm, rotated rx 180 ry 0 rz 180 deg; joints [-137.415, -53.452, -95.633, 46.97, 67.773, -22.059]
  MoveL 4875 to (-37.63, 41.3, 78.65) mm, rotated rx 180 ry 0 rz 180 deg; joints [-137.415, -53.452, -95.633, 46.97, 67.773, -22.059]
  Call Extruder(66.57570)
  MoveL 4876 to (-37.3, 40.85, 78.65) mm, rotated rx -180 ry 0 rz -180 deg; joints [-137.506, -53.449, -95.644, 46.877, 67.744, -22.019]
  Call Extruder(67.40363)
  MoveL 4877 to (-36.39, 39.81, 78.65) mm, rotated rx 180 ry 0 rz -180 deg; joints [-137.733, -53.448, -95.648, 46.649, 67.661, -21.93]
  Call Extruder(68.23154)
  MoveL 4878 to (-35.35, 38.9, 78.65) mm, rotated rx 180 ry 0 rz -180 deg; joints [-137.958, -53.456, -95.621, 46.428, 67.565, -21.858]
  Call Extruder(68.39885)
  MoveL 4879 to (-35.13, 38.73, 78.65) mm, rotated rx -180 ry 0 rz 180 deg; joints [-138.003, -53.459, -95.612, 46.385, 67.543, -21.847]
  MoveL 4880 to (-35.13, 38.73, 78.65) mm, rotated rx -180 ry 0 rz 180 deg; joints [-138.003, -53.459, -95.612, 46.385, 67.543, -21.847]
  Call Extruder(68.73227)
  MoveL 4881 to (-34.68, 38.41, 78.65) mm, rotated rx 180 ry 0 rz 180 deg; joints [-138.092, -53.465, -95.592, 46.299, 67.501, -21.823]
  MoveL 4882 to (-34.68, 38.41, 78.65) mm, rotated rx 180 ry 0 rz 180 deg; joints [-138.092, -53.465, -95.592, 46.299, 67.501, -21.823]
  Call Extruder(69.06451)
  MoveL 4883 to (-34.22, 38.08, 78.65) mm, rotated rx 180 ry 0 rz -180 deg; joints [-138.182, -53.471, -95.572, 46.213, 67.458, -21.799]
  MoveL 4884 to (-34.22, 38.08, 78.65) mm, rotated rx 180 ry 0 rz -180 deg; joints [-138.182, -53.471, -95.572, 46.213, 67.458, -21.799]
  Call Extruder(69.18222)
  MoveL 4885 to (-34.05, 37.98, 78.65) mm, rotated rx 180 ry 0 rz 180 deg; joints [-138.213, -53.474, -95.562, 46.185, 67.442, -21.793]
  MoveL 4886 to (-34.05, 37.98, 78.65) mm, rotated rx 180 ry 0 rz 180 deg; joints [-138.213, -53.474, -95.562, 46.185, 67.442, -21.793]
  Call Extruder(69.38994)
  MoveL 4887 to (-33.75, 37.8, 78.65) mm, rotated rx 180 ry 0 rz 180 deg; joints [-138.267, -53.48, -95.543, 46.134, 67.412, -21.782]
  MoveL 4888 to (-33.75, 37.8, 78.65) mm, rotated rx 180 ry 0 rz 180 deg; joints [-138.267, -53.48, -95.543, 46.134, 67.412, -21.782]
  Call Extruder(69.59688)
  MoveL 4889 to (-33.45, 37.63, 78.65) mm, rotated rx -180 ry 0 rz -180 deg; joints [-138.322, -53.486, -95.525, 46.083, 67.383, -21.771]
  MoveL 4890 to (-33.45, 37.63, 78.65) mm, rotated rx -180 ry 0 rz -180 deg; joints [-138.322, -53.486, -95.525, 46.083, 67.383, -21.771]
  Call Extruder(69.80304)
  MoveL 4891 to (-33.14, 37.45, 78.65) mm, rotated rx -180 ry 0 rz 180 deg; joints [-138.376, -53.491, -95.506, 46.032, 67.354, -21.76]
  MoveL 4892 to (-33.14, 37.45, 78.65) mm, rotated rx -180 ry 0 rz 180 deg; joints [-138.376, -53.491, -95.506, 46.032, 67.354, -21.76]
  Call Extruder(69.98473)
  MoveL 4893 to (-32.87, 37.31, 78.65) mm, rotated rx 180 ry 0 rz 180 deg; joints [-138.424, -53.497, -95.487, 45.988, 67.327, -21.751]
  MoveL 4894 to (-32.87, 37.31, 78.65) mm, rotated rx 180 ry 0 rz 180 deg; joints [-138.424, -53.497, -95.487, 45.988, 67.327, -21.751]
  Call Extruder(70.14273)
  MoveL 4895 to (-32.62, 37.2, 78.65) mm, rotated rx 180 ry 0 rz -180 deg; joints [-138.464, -53.503, -95.467, 45.951, 67.303, -21.746]
  MoveL 4896 to (-32.62, 37.2, 78.65) mm, rotated rx 180 ry 0 rz -180 deg; joints [-138.464, -53.503, -95.467, 45.951, 67.303, -21.746]
  Call Extruder(70.30013)
  MoveL 4897 to (-32.37, 37.09, 78.65) mm, rotated rx 180 ry 0 rz 180 deg; joints [-138.504, -53.509, -95.448, 45.915, 67.279, -21.741]
  MoveL 4898 to (-32.37, 37.09, 78.65) mm, rotated rx 180 ry 0 rz 180 deg; joints [-138.504, -53.509, -95.448, 45.915, 67.279, -21.741]
  Call Extruder(70.48284)
  MoveL 4899 to (-32.08, 36.97, 78.65) mm, rotated rx 180 ry 0 rz 180 deg; joints [-138.551, -53.517, -95.424, 45.873, 67.25, -21.736]
  MoveL 4900 to (-32.08, 36.97, 78.65) mm, rotated rx 180 ry 0 rz 180 deg; joints [-138.551, -53.517, -95.424, 45.873, 67.25, -21.736]
  Call Extruder(70.66479)
  MoveL 4901 to (-31.78, 36.85, 78.65) mm, rotated rx 180 ry 0 rz 180 deg; joints [-138.597, -53.524, -95.401, 45.831, 67.222, -21.73]
  MoveL 4902 to (-31.78, 36.85, 78.65) mm, rotated rx 180 ry 0 rz 180 deg; joints [-138.597, -53.524, -95.401, 45.831, 67.222, -21.73]
  Call Extruder(70.81212)
  MoveL 4903 to (-31.54, 36.76, 78.65) mm, rotated rx 180 ry 0 rz 180 deg; joints [-138.634, -53.53, -95.38, 45.798, 67.198, -21.727]
  MoveL 4904 to (-31.54, 36.76, 78.65) mm, rotated rx 180 ry 0 rz 180 deg; joints [-138.634, -53.53, -95.38, 45.798, 67.198, -21.727]
  Call Extruder(70.92535)
  MoveL 4905 to (-31.35, 36.7, 78.65) mm, rotated rx -180 ry 0 rz -180 deg; joints [-138.662, -53.536, -95.363, 45.773, 67.18, -21.725]
  MoveL 4906 to (-31.35, 36.7, 78.65) mm, rotated rx -180 ry 0 rz -180 deg; joints [-138.662, -53.536, -95.363, 45.773, 67.18, -21.725]
  Call Extruder(71.03815)
  MoveL 4907 to (-31.17, 36.64, 78.65) mm, rotated rx 180 ry 0 rz 180 deg; joints [-138.69, -53.541, -95.346, 45.749, 67.161, -21.723]
  MoveL 4908 to (-31.17, 36.64, 78.65) mm, rotated rx 180 ry 0 rz 180 deg; joints [-138.69, -53.541, -95.346, 45.749, 67.161, -21.723]
  Call Extruder(71.15049)
  MoveL 4909 to (-30.98, 36.58, 78.65) mm, rotated rx -180 ry 0 rz 180 deg; joints [-138.718, -53.546, -95.329, 45.725, 67.143, -21.722]
  MoveL 4910 to (-30.98, 36.58, 78.65) mm, rotated rx -180 ry 0 rz 180 deg; joints [-138.718, -53.546, -95.329, 45.725, 67.143, -21.722]
  Call Extruder(71.26240)
  MoveL 4911 to (-30.79, 36.52, 78.65) mm, rotated rx -180 ry 0 rz 180 deg; joints [-138.745, -53.552, -95.312, 45.7, 67.124, -21.72]
  MoveL 4912 to (-30.79, 36.52, 78.65) mm, rotated rx -180 ry 0 rz 180 deg; joints [-138.745, -53.552, -95.312, 45.7, 67.124, -21.72]
  Call Extruder(71.38380)
  MoveL 4913 to (-30.58, 36.45, 78.65) mm, rotated rx -180 ry 0 rz 180 deg; joints [-138.776, -53.558, -95.293, 45.674, 67.104, -21.718]
  MoveL 4914 to (-30.58, 36.45, 78.65) mm, rotated rx -180 ry 0 rz 180 deg; joints [-138.776, -53.558, -95.293, 45.674, 67.104, -21.718]
  Call Extruder(71.51459)
  MoveL 4915 to (-30.36, 36.39, 78.65) mm, rotated rx 180 ry 0 rz 180 deg; joints [-138.808, -53.564, -95.272, 45.645, 67.082, -21.717]
  MoveL 4916 to (-30.36, 36.39, 78.65) mm, rotated rx 180 ry 0 rz 180 deg; joints [-138.808, -53.564, -95.272, 45.645, 67.082, -21.717]
  Call Extruder(71.64481)
  MoveL 4917 to (-30.14, 36.32, 78.65) mm, rotated rx 180 ry 0 rz 180 deg; joints [-138.84, -53.571, -95.251, 45.617, 67.06, -21.715]
  MoveL 4918 to (-30.14, 36.32, 78.65) mm, rotated rx 180 ry 0 rz 180 deg; joints [-138.84, -53.571, -95.251, 45.617, 67.06, -21.715]
  Call Extruder(71.77447)
  MoveL 4919 to (-29.91, 36.25, 78.65) mm, rotated rx 180 ry 0 rz -180 deg; joints [-138.873, -53.577, -95.23, 45.589, 67.038, -21.714]
  MoveL 4920 to (-29.91, 36.25, 78.65) mm, rotated rx 180 ry 0 rz -180 deg; joints [-138.873, -53.577, -95.23, 45.589, 67.038, -21.714]
  Call Extruder(71.90357)
  MoveL 4921 to (-29.69, 36.18, 78.65) mm, rotated rx 180 ry 0 rz -180 deg; joints [-138.905, -53.584, -95.209, 45.561, 67.016, -21.712]
  MoveL 4922 to (-29.69, 36.18, 78.65) mm, rotated rx 180 ry 0 rz -180 deg; joints [-138.905, -53.584, -95.209, 45.561, 67.016, -21.712]
  Call Extruder(72.01864)
  MoveL 4923 to (-29.48, 36.14, 78.65) mm, rotated rx 180 ry 0 rz -180 deg; joints [-138.932, -53.59, -95.188, 45.538, 66.995, -21.713]
  MoveL 4924 to (-29.48, 36.14, 78.65) mm, rotated rx 180 ry 0 rz -180 deg; joints [-138.932, -53.59, -95.188, 45.538, 66.995, -21.713]
  Call Extruder(72.13326)
  MoveL 4925 to (-29.28, 36.09, 78.65) mm, rotated rx 180 ry 0 rz 180 deg; joints [-138.96, -53.597, -95.167, 45.514, 66.975, -21.713]
  MoveL 4926 to (-29.28, 36.09, 78.65) mm, rotated rx 180 ry 0 rz 180 deg; joints [-138.96, -53.597, -95.167, 45.514, 66.975, -21.713]
  Call Extruder(72.24743)
  MoveL 4927 to (-29.08, 36.05, 78.65) mm, rotated rx 180 ry 0 rz -180 deg; joints [-138.987, -53.603, -95.145, 45.491, 66.955, -21.714]
  MoveL 4928 to (-29.08, 36.05, 78.65) mm, rotated rx 180 ry 0 rz -180 deg; joints [-138.987, -53.603, -95.145, 45.491, 66.955, -21.714]
  Call Extruder(72.36115)
  MoveL 4929 to (-28.87, 36, 78.65) mm, rotated rx 180 ry 0 rz 180 deg; joints [-139.014, -53.61, -95.124, 45.468, 66.934, -21.714]
  MoveL 4930 to (-28.87, 36, 78.65) mm, rotated rx 180 ry 0 rz 180 deg; joints [-139.014, -53.61, -95.124, 45.468, 66.934, -21.714]
  Call Extruder(72.48657)
  MoveL 4931 to (-28.64, 35.96, 78.65) mm, rotated rx 180 ry 0 rz 180 deg; joints [-139.044, -53.617, -95.101, 45.443, 66.912, -21.715]
  MoveL 4932 to (-28.64, 35.96, 78.65) mm, rotated rx 180 ry 0 rz 180 deg; joints [-139.044, -53.617, -95.101, 45.443, 66.912, -21.715]
  Call Extruder(72.62355)
  MoveL 4933 to (-28.4, 35.91, 78.65) mm, rotated rx -180 ry 0 rz -180 deg; joints [-139.077, -53.626, -95.074, 45.415, 66.887, -21.716]
  MoveL 4934 to (-28.4, 35.91, 78.65) mm, rotated rx -180 ry 0 rz -180 deg; joints [-139.077, -53.626, -95.074, 45.415, 66.887, -21.716]
  Call Extruder(72.75991)
  MoveL 4935 to (-28.15, 35.86, 78.65) mm, rotated rx -180 ry 0 rz -180 deg; joints [-139.109, -53.634, -95.048, 45.388, 66.862, -21.717]
  MoveL 4936 to (-28.15, 35.86, 78.65) mm, rotated rx -180 ry 0 rz -180 deg; joints [-139.109, -53.634, -95.048, 45.388, 66.862, -21.717]
  Call Extruder(72.89567)
  MoveL 4937 to (-27.9, 35.81, 78.65) mm, rotated rx 180 ry 0 rz 180 deg; joints [-139.142, -53.642, -95.021, 45.361, 66.837, -21.719]
  MoveL 4938 to (-27.9, 35.81, 78.65) mm, rotated rx 180 ry 0 rz 180 deg; joints [-139.142, -53.642, -95.021, 45.361, 66.837, -21.719]
  Call Extruder(73.03082)
  MoveL 4939 to (-27.65, 35.76, 78.65) mm, rotated rx 180 ry 0 rz 180 deg; joints [-139.174, -53.651, -94.995, 45.333, 66.813, -21.72]
  MoveL 4940 to (-27.65, 35.76, 78.65) mm, rotated rx 180 ry 0 rz 180 deg; joints [-139.174, -53.651, -94.995, 45.333, 66.813, -21.72]
  Call Extruder(73.16535)
  MoveL 4941 to (-27.4, 35.71, 78.65) mm, rotated rx 180 ry 0 rz -180 deg; joints [-139.207, -53.659, -94.968, 45.306, 66.788, -21.721]
  MoveL 4942 to (-27.4, 35.71, 78.65) mm, rotated rx 180 ry 0 rz -180 deg; joints [-139.207, -53.659, -94.968, 45.306, 66.788, -21.721]
  Call Extruder(73.29928)
  MoveL 4943 to (-27.15, 35.66, 78.65) mm, rotated rx 180 ry 0 rz -180 deg; joints [-139.239, -53.667, -94.942, 45.279, 66.763, -21.722]
  MoveL 4944 to (-27.15, 35.66, 78.65) mm, rotated rx 180 ry 0 rz -180 deg; joints [-139.239, -53.667, -94.942, 45.279, 66.763, -21.722]
  Call Extruder(73.44714)
  MoveL 4945 to (-26.87, 35.61, 78.65) mm, rotated rx 180 ry 0 rz -180 deg; joints [-139.275, -53.677, -94.911, 45.249, 66.735, -21.724]
  MoveL 4946 to (-26.87, 35.61, 78.65) mm, rotated rx 180 ry 0 rz -180 deg; joints [-139.275, -53.677, -94.911, 45.249, 66.735, -21.724]
  Call Extruder(73.60887)
  MoveL 4947 to (-26.57, 35.56, 78.65) mm, rotated rx 180 ry 0 rz -180 deg; joints [-139.313, -53.687, -94.877, 45.218, 66.705, -21.727]
  MoveL 4948 to (-26.57, 35.56, 78.65) mm, rotated rx 180 ry 0 rz -180 deg; joints [-139.313, -53.687, -94.877, 45.218, 66.705, -21.727]
  Call Extruder(73.76988)
  MoveL 4949 to (-26.26, 35.51, 78.65) mm, rotated rx -180 ry 0 rz 180 deg; joints [-139.351, -53.698, -94.843, 45.186, 66.674, -21.729]
  MoveL 4950 to (-26.26, 35.51, 78.65) mm, rotated rx -180 ry 0 rz 180 deg; joints [-139.351, -53.698, -94.843, 45.186, 66.674, -21.729]
  Call Extruder(73.93016)
  MoveL 4951 to (-25.96, 35.46, 78.65) mm, rotated rx -180 ry 0 rz 180 deg; joints [-139.39, -53.709, -94.809, 45.155, 66.643, -21.732]
  MoveL 4952 to (-25.96, 35.46, 78.65) mm, rotated rx -180 ry 0 rz 180 deg; joints [-139.39, -53.709, -94.809, 45.155, 66.643, -21.732]
  Call Extruder(74.08971)
  MoveL 4953 to (-25.65, 35.42, 78.65) mm, rotated rx 180 ry 0 rz 180 deg; joints [-139.428, -53.719, -94.775, 45.123, 66.613, -21.735]
  MoveL 4954 to (-25.65, 35.42, 78.65) mm, rotated rx 180 ry 0 rz 180 deg; joints [-139.428, -53.719, -94.775, 45.123, 66.613, -21.735]
  Call Extruder(74.24853)
  MoveL 4955 to (-25.34, 35.37, 78.65) mm, rotated rx -180 ry 0 rz 180 deg; joints [-139.466, -53.73, -94.741, 45.092, 66.582, -21.738]
  MoveL 4956 to (-25.34, 35.37, 78.65) mm, rotated rx -180 ry 0 rz 180 deg; joints [-139.466, -53.73, -94.741, 45.092, 66.582, -21.738]
  Call Extruder(74.42720)
  MoveL 4957 to (-25, 35.32, 78.65) mm, rotated rx 180 ry 0 rz -180 deg; joints [-139.508, -53.743, -94.701, 45.057, 66.547, -21.742]
  MoveL 4958 to (-25, 35.32, 78.65) mm, rotated rx 180 ry 0 rz -180 deg; joints [-139.508, -53.743, -94.701, 45.057, 66.547, -21.742]
  Call Extruder(74.62564)
  MoveL 4959 to (-24.61, 35.27, 78.65) mm, rotated rx -180 ry 0 rz 180 deg; joints [-139.554, -53.757, -94.656, 45.02, 66.508, -21.747]
  MoveL 4960 to (-24.61, 35.27, 78.65) mm, rotated rx -180 ry 0 rz 180 deg; joints [-139.554, -53.757, -94.656, 45.02, 66.508, -21.747]
  Call Extruder(74.82322)
  MoveL 4961 to (-24.22, 35.23, 78.65) mm, rotated rx 180 ry 0 rz -180 deg; joints [-139.6, -53.771, -94.611, 44.983, 66.469, -21.752]
  MoveL 4962 to (-24.22, 35.23, 78.65) mm, rotated rx 180 ry 0 rz -180 deg; joints [-139.6, -53.771, -94.611, 44.983, 66.469, -21.752]
  Call Extruder(75.01993)
  MoveL 4963 to (-23.84, 35.18, 78.65) mm, rotated rx 180 ry 0 rz 180 deg; joints [-139.647, -53.785, -94.566, 44.946, 66.43, -21.757]
  MoveL 4964 to (-23.84, 35.18, 78.65) mm, rotated rx 180 ry 0 rz 180 deg; joints [-139.647, -53.785, -94.566, 44.946, 66.43, -21.757]
  Call Extruder(75.21577)
  MoveL 4965 to (-23.45, 35.14, 78.65) mm, rotated rx -180 ry 0 rz 180 deg; joints [-139.693, -53.8, -94.521, 44.909, 66.391, -21.762]
  MoveL 4966 to (-23.45, 35.14, 78.65) mm, rotated rx -180 ry 0 rz 180 deg; joints [-139.693, -53.8, -94.521, 44.909, 66.391, -21.762]
  Call Extruder(75.51116)
  MoveL 4967 to (-22.86, 35.09, 78.65) mm, rotated rx 180 ry 0 rz 180 deg; joints [-139.76, -53.822, -94.449, 44.856, 66.332, -21.773]
  MoveL 4968 to (-22.86, 35.09, 78.65) mm, rotated rx 180 ry 0 rz 180 deg; joints [-139.76, -53.822, -94.449, 44.856, 66.332, -21.773]
  Call Extruder(75.80522)
  MoveL 4969 to (-22.27, 35.05, 78.65) mm, rotated rx 180 ry 0 rz -180 deg; joints [-139.826, -53.845, -94.377, 44.803, 66.272, -21.783]
  MoveL 4970 to (-22.27, 35.05, 78.65) mm, rotated rx 180 ry 0 rz -180 deg; joints [-139.826, -53.845, -94.377, 44.803, 66.272, -21.783]
  Call Extruder(76.09795)
  MoveL 4971 to (-21.68, 35, 78.65) mm, rotated rx 180 ry 0 rz 180 deg; joints [-139.893, -53.868, -94.306, 44.75, 66.213, -21.794]
  MoveL 4972 to (-21.68, 35, 78.65) mm, rotated rx 180 ry 0 rz 180 deg; joints [-139.893, -53.868, -94.306, 44.75, 66.213, -21.794]
  Call Extruder(76.67140)
  MoveL 4973 to (-20.52, 34.95, 78.65) mm, rotated rx 180 ry 0 rz -180 deg; joints [-140.019, -53.914, -94.159, 44.654, 66.095, -21.819]
  MoveL 4974 to (-20.52, 34.95, 78.65) mm, rotated rx 180 ry 0 rz -180 deg; joints [-140.019, -53.914, -94.159, 44.654, 66.095, -21.819]
  Call Extruder(77.38537)
  MoveL 4975 to (-19.06, 34.91, 78.65) mm, rotated rx 180 ry 0 rz 180 deg; joints [-140.173, -53.974, -93.972, 44.537, 65.947, -21.853]
  Call Extruder(194.23211)
  MoveL 4976 to (219.06, 34.91, 78.65) mm, rotated rx -180 ry 0 rz -180 deg; joints [-155.896, -71.139, -51.523, 39.659, 39.784, -32.5]
  Call Extruder(194.66067)
  MoveL 4977 to (219.94, 34.93, 78.65) mm, rotated rx 180 ry 0 rz -180 deg; joints [-155.931, -71.239, -51.306, 39.703, 39.675, -32.582]
  MoveL 4978 to (219.94, 34.93, 78.65) mm, rotated rx 180 ry 0 rz -180 deg; joints [-155.931, -71.239, -51.306, 39.703, 39.675, -32.582]
  Call Extruder(195.23412)
  MoveL 4979 to (221.1, 34.97, 78.65) mm, rotated rx 180 ry 0 rz 180 deg; joints [-155.975, -71.372, -51.015, 39.767, 39.53, -32.695]
  MoveL 4980 to (221.1, 34.97, 78.65) mm, rotated rx 180 ry 0 rz 180 deg; joints [-155.975, -71.372, -51.015, 39.767, 39.53, -32.695]
  Call Extruder(195.66843)
  MoveL 4981 to (221.97, 35.02, 78.65) mm, rotated rx 180 ry 0 rz 180 deg; joints [-156.007, -71.474, -50.793, 39.818, 39.421, -32.783]
  MoveL 4982 to (221.97, 35.02, 78.65) mm, rotated rx 180 ry 0 rz 180 deg; joints [-156.007, -71.474, -50.793, 39.818, 39.421, -32.783]
  Call Extruder(195.96249)
  MoveL 4983 to (222.56, 35.07, 78.65) mm, rotated rx 180 ry 0 rz 180 deg; joints [-156.027, -71.544, -50.642, 39.855, 39.347, -32.845]
  MoveL 4984 to (222.56, 35.07, 78.65) mm, rotated rx 180 ry 0 rz 180 deg; joints [-156.027, -71.544, -50.642, 39.855, 39.347, -32.845]
  Call Extruder(196.25788)
  MoveL 4985 to (223.15, 35.11, 78.65) mm, rotated rx 180 ry 0 rz 180 deg; joints [-156.047, -71.614, -50.49, 39.893, 39.273, -32.908]
  MoveL 4986 to (223.15, 35.11, 78.65) mm, rotated rx 180 ry 0 rz 180 deg; joints [-156.047, -71.614, -50.49, 39.893, 39.273, -32.908]
  Call Extruder(196.50411)
  MoveL 4987 to (223.64, 35.16, 78.65) mm, rotated rx -180 ry 0 rz 180 deg; joints [-156.062, -71.672, -50.363, 39.926, 39.212, -32.961]
  MoveL 4988 to (223.64, 35.16, 78.65) mm, rotated rx -180 ry 0 rz 180 deg; joints [-156.062, -71.672, -50.363, 39.926, 39.212, -32.961]
  Call Extruder(196.70082)
  MoveL 4989 to (224.03, 35.21, 78.65) mm, rotated rx -180 ry 0 rz 180 deg; joints [-156.074, -71.719, -50.261, 39.954, 39.164, -33.005]
  MoveL 4990 to (224.03, 35.21, 78.65) mm, rotated rx -180 ry 0 rz 180 deg; joints [-156.074, -71.719, -50.261, 39.954, 39.164, -33.005]
  Call Extruder(196.89839)
  MoveL 4991 to (224.42, 35.25, 78.65) mm, rotated rx 180 ry 0 rz 180 deg; joints [-156.086, -71.766, -50.16, 39.982, 39.115, -33.049]
  MoveL 4992 to (224.42, 35.25, 78.65) mm, rotated rx 180 ry 0 rz 180 deg; joints [-156.086, -71.766, -50.16, 39.982, 39.115, -33.049]
  Call Extruder(197.09684)
  MoveL 4993 to (224.8, 35.3, 78.65) mm, rotated rx 180 ry 0 rz 180 deg; joints [-156.097, -71.813, -50.057, 40.01, 39.067, -33.093]
  MoveL 4994 to (224.8, 35.3, 78.65) mm, rotated rx 180 ry 0 rz 180 deg; joints [-156.097, -71.813, -50.057, 40.01, 39.067, -33.093]
  Call Extruder(197.29615)
  MoveL 4995 to (225.19, 35.34, 78.65) mm, rotated rx -180 ry 0 rz 180 deg; joints [-156.109, -71.86, -49.955, 40.038, 39.018, -33.137]
  MoveL 4996 to (225.19, 35.34, 78.65) mm, rotated rx -180 ry 0 rz 180 deg; joints [-156.109, -71.86, -49.955, 40.038, 39.018, -33.137]
  Call Extruder(197.45497)
  MoveL 4997 to (225.5, 35.39, 78.65) mm, rotated rx -180 ry 0 rz 180 deg; joints [-156.117, -71.898, -49.873, 40.063, 38.98, -33.174]
  MoveL 4998 to (225.5, 35.39, 78.65) mm, rotated rx -180 ry 0 rz 180 deg; joints [-156.117, -71.898, -49.873, 40.063, 38.98, -33.174]
  Call Extruder(197.61451)
  MoveL 4999 to (225.8, 35.44, 78.65) mm, rotated rx -180 ry 0 rz 180 deg; joints [-156.125, -71.936, -49.79, 40.087, 38.942, -33.211]
  MoveL 5000 to (225.8, 35.44, 78.65) mm, rotated rx -180 ry 0 rz 180 deg; joints [-156.125, -71.936, -49.79, 40.087, 38.942, -33.211]
  Call Extruder(197.77479)
  MoveL 5001 to (226.11, 35.49, 78.65) mm, rotated rx 180 ry 0 rz -180 deg; joints [-156.133, -71.974, -49.708, 40.112, 38.903, -33.248]
  MoveL 5002 to (226.11, 35.49, 78.65) mm, rotated rx 180 ry 0 rz -180 deg; joints [-156.133, -71.974, -49.708, 40.112, 38.903, -33.248]
  Call Extruder(197.93579)
  MoveL 5003 to (226.41, 35.54, 78.65) mm, rotated rx -180 ry 0 rz -180 deg; joints [-156.141, -72.012, -49.626, 40.137, 38.865, -33.286]
  MoveL 5004 to (226.41, 35.54, 78.65) mm, rotated rx -180 ry 0 rz -180 deg; joints [-156.141, -72.012, -49.626, 40.137, 38.865, -33.286]
  Call Extruder(198.09752)
  MoveL 5005 to (226.72, 35.59, 78.65) mm, rotated rx 180 ry 0 rz 180 deg; joints [-156.149, -72.05, -49.543, 40.162, 38.827, -33.323]
  MoveL 5006 to (226.72, 35.59, 78.65) mm, rotated rx 180 ry 0 rz 180 deg; joints [-156.149, -72.05, -49.543, 40.162, 38.827, -33.323]
  Call Extruder(198.25998)
  MoveL 5007 to (227.02, 35.63, 78.65) mm, rotated rx 180 ry 0 rz 180 deg; joints [-156.157, -72.088, -49.46, 40.187, 38.788, -33.361]
  MoveL 5008 to (227.02, 35.63, 78.65) mm, rotated rx 180 ry 0 rz 180 deg; joints [-156.157, -72.088, -49.46, 40.187, 38.788, -33.361]
  Call Extruder(198.39391)
  MoveL 5009 to (227.27, 35.68, 78.65) mm, rotated rx 180 ry 0 rz 180 deg; joints [-156.162, -72.12, -49.392, 40.209, 38.757, -33.393]
  MoveL 5010 to (227.27, 35.68, 78.65) mm, rotated rx 180 ry 0 rz 180 deg; joints [-156.162, -72.12, -49.392, 40.209, 38.757, -33.393]
  Call Extruder(198.52845)
  MoveL 5011 to (227.52, 35.73, 78.65) mm, rotated rx 180 ry 0 rz 180 deg; joints [-156.168, -72.152, -49.323, 40.232, 38.726, -33.425]
  MoveL 5012 to (227.52, 35.73, 78.65) mm, rotated rx 180 ry 0 rz 180 deg; joints [-156.168, -72.152, -49.323, 40.232, 38.726, -33.425]
  Call Extruder(198.66359)
  MoveL 5013 to (227.77, 35.78, 78.65) mm, rotated rx -180 ry 0 rz 180 deg; joints [-156.173, -72.183, -49.254, 40.254, 38.694, -33.458]
  MoveL 5014 to (227.77, 35.78, 78.65) mm, rotated rx -180 ry 0 rz 180 deg; joints [-156.173, -72.183, -49.254, 40.254, 38.694, -33.458]
  Call Extruder(198.79935)
  MoveL 5015 to (228.02, 35.83, 78.65) mm, rotated rx -180 ry 0 rz 180 deg; joints [-156.179, -72.215, -49.186, 40.276, 38.663, -33.49]
  MoveL 5016 to (228.02, 35.83, 78.65) mm, rotated rx -180 ry 0 rz 180 deg; joints [-156.179, -72.215, -49.186, 40.276, 38.663, -33.49]
  Call Extruder(198.93572)
  MoveL 5017 to (228.27, 35.88, 78.65) mm, rotated rx 180 ry 0 rz 180 deg; joints [-156.185, -72.247, -49.117, 40.299, 38.632, -33.523]
  MoveL 5018 to (228.27, 35.88, 78.65) mm, rotated rx 180 ry 0 rz 180 deg; joints [-156.185, -72.247, -49.117, 40.299, 38.632, -33.523]
  Call Extruder(199.07270)
  MoveL 5019 to (228.52, 35.93, 78.65) mm, rotated rx 180 ry 0 rz -180 deg; joints [-156.19, -72.279, -49.048, 40.322, 38.601, -33.555]
  MoveL 5020 to (228.52, 35.93, 78.65) mm, rotated rx 180 ry 0 rz -180 deg; joints [-156.19, -72.279, -49.048, 40.322, 38.601, -33.555]
  Call Extruder(199.21029)
  MoveL 5021 to (228.77, 35.98, 78.65) mm, rotated rx 180 ry 0 rz -180 deg; joints [-156.196, -72.311, -48.979, 40.344, 38.569, -33.588]
  MoveL 5022 to (228.77, 35.98, 78.65) mm, rotated rx 180 ry 0 rz -180 deg; joints [-156.196, -72.311, -48.979, 40.344, 38.569, -33.588]
  Call Extruder(199.32400)
  MoveL 5023 to (228.97, 36.03, 78.65) mm, rotated rx -180 ry 0 rz 180 deg; joints [-156.2, -72.337, -48.922, 40.364, 38.544, -33.616]
  MoveL 5024 to (228.97, 36.03, 78.65) mm, rotated rx -180 ry 0 rz 180 deg; joints [-156.2, -72.337, -48.922, 40.364, 38.544, -33.616]
  Call Extruder(199.43818)
  MoveL 5025 to (229.18, 36.07, 78.65) mm, rotated rx -180 ry 0 rz 180 deg; joints [-156.204, -72.364, -48.864, 40.383, 38.518, -33.643]
  MoveL 5026 to (229.18, 36.07, 78.65) mm, rotated rx -180 ry 0 rz 180 deg; joints [-156.204, -72.364, -48.864, 40.383, 38.518, -33.643]
  Call Extruder(199.55280)
  MoveL 5027 to (229.38, 36.12, 78.65) mm, rotated rx -180 ry 0 rz 180 deg; joints [-156.208, -72.39, -48.807, 40.403, 38.492, -33.671]
  MoveL 5028 to (229.38, 36.12, 78.65) mm, rotated rx -180 ry 0 rz 180 deg; joints [-156.208, -72.39, -48.807, 40.403, 38.492, -33.671]
  Call Extruder(199.66788)
  MoveL 5029 to (229.59, 36.16, 78.65) mm, rotated rx 180 ry 0 rz 180 deg; joints [-156.212, -72.417, -48.75, 40.422, 38.466, -33.699]
  MoveL 5030 to (229.59, 36.16, 78.65) mm, rotated rx 180 ry 0 rz 180 deg; joints [-156.212, -72.417, -48.75, 40.422, 38.466, -33.699]
  Call Extruder(199.79011)
  MoveL 5031 to (229.8, 36.22, 78.65) mm, rotated rx 180 ry 0 rz 180 deg; joints [-156.216, -72.445, -48.689, 40.444, 38.44, -33.729]
  MoveL 5032 to (229.8, 36.22, 78.65) mm, rotated rx 180 ry 0 rz 180 deg; joints [-156.216, -72.445, -48.689, 40.444, 38.44, -33.729]
  Call Extruder(199.91978)
  MoveL 5033 to (230.02, 36.28, 78.65) mm, rotated rx 180 ry 0 rz -180 deg; joints [-156.219, -72.475, -48.624, 40.469, 38.411, -33.763]
  MoveL 5034 to (230.02, 36.28, 78.65) mm, rotated rx 180 ry 0 rz -180 deg; joints [-156.219, -72.475, -48.624, 40.469, 38.411, -33.763]
  Call Extruder(200.05001)
  MoveL 5035 to (230.25, 36.35, 78.65) mm, rotated rx -180 ry 0 rz 180 deg; joints [-156.221, -72.505, -48.559, 40.494, 38.383, -33.796]
  MoveL 5036 to (230.25, 36.35, 78.65) mm, rotated rx -180 ry 0 rz 180 deg; joints [-156.221, -72.505, -48.559, 40.494, 38.383, -33.796]
  Call Extruder(200.18080)
  MoveL 5037 to (230.47, 36.42, 78.65) mm, rotated rx 180 ry 0 rz 180 deg; joints [-156.224, -72.535, -48.494, 40.519, 38.355, -33.83]
  MoveL 5038 to (230.47, 36.42, 78.65) mm, rotated rx 180 ry 0 rz 180 deg; joints [-156.224, -72.535, -48.494, 40.519, 38.355, -33.83]
  Call Extruder(200.31217)
  MoveL 5039 to (230.69, 36.49, 78.65) mm, rotated rx 180 ry 0 rz 180 deg; joints [-156.227, -72.566, -48.429, 40.544, 38.327, -33.863]
  MoveL 5040 to (230.69, 36.49, 78.65) mm, rotated rx 180 ry 0 rz 180 deg; joints [-156.227, -72.566, -48.429, 40.544, 38.327, -33.863]
  Call Extruder(200.42119)
  MoveL 5041 to (230.88, 36.55, 78.65) mm, rotated rx 180 ry 0 rz 180 deg; joints [-156.229, -72.59, -48.375, 40.565, 38.304, -33.892]
  MoveL 5042 to (230.88, 36.55, 78.65) mm, rotated rx 180 ry 0 rz 180 deg; joints [-156.229, -72.59, -48.375, 40.565, 38.304, -33.892]
  Call Extruder(200.53270)
  MoveL 5043 to (231.06, 36.61, 78.65) mm, rotated rx 180 ry 0 rz -180 deg; joints [-156.231, -72.616, -48.32, 40.586, 38.281, -33.92]
  MoveL 5044 to (231.06, 36.61, 78.65) mm, rotated rx 180 ry 0 rz -180 deg; joints [-156.231, -72.616, -48.32, 40.586, 38.281, -33.92]
  Call Extruder(200.64671)
  MoveL 5045 to (231.26, 36.67, 78.65) mm, rotated rx 180 ry 0 rz 180 deg; joints [-156.233, -72.642, -48.264, 40.609, 38.256, -33.95]
  MoveL 5046 to (231.26, 36.67, 78.65) mm, rotated rx 180 ry 0 rz 180 deg; joints [-156.233, -72.642, -48.264, 40.609, 38.256, -33.95]
  Call Extruder(200.76118)
  MoveL 5047 to (231.45, 36.73, 78.65) mm, rotated rx 180 ry 0 rz -180 deg; joints [-156.235, -72.668, -48.207, 40.631, 38.232, -33.98]
  MoveL 5048 to (231.45, 36.73, 78.65) mm, rotated rx 180 ry 0 rz -180 deg; joints [-156.235, -72.668, -48.207, 40.631, 38.232, -33.98]
  Call Extruder(200.87611)
  MoveL 5049 to (231.64, 36.79, 78.65) mm, rotated rx 180 ry 0 rz 180 deg; joints [-156.237, -72.694, -48.151, 40.653, 38.209, -34.009]
  MoveL 5050 to (231.64, 36.79, 78.65) mm, rotated rx 180 ry 0 rz 180 deg; joints [-156.237, -72.694, -48.151, 40.653, 38.209, -34.009]
  Call Extruder(201.05806)
  MoveL 5051 to (231.93, 36.91, 78.65) mm, rotated rx 180 ry 0 rz 180 deg; joints [-156.238, -72.736, -48.062, 40.692, 38.172, -34.059]
  MoveL 5052 to (231.93, 36.91, 78.65) mm, rotated rx 180 ry 0 rz 180 deg; joints [-156.238, -72.736, -48.062, 40.692, 38.172, -34.059]
  Call Extruder(201.24078)
  MoveL 5053 to (232.22, 37.03, 78.65) mm, rotated rx -180 ry 0 rz 180 deg; joints [-156.238, -72.777, -47.973, 40.73, 38.135, -34.109]
  MoveL 5054 to (232.22, 37.03, 78.65) mm, rotated rx -180 ry 0 rz 180 deg; joints [-156.238, -72.777, -47.973, 40.73, 38.135, -34.109]
  Call Extruder(201.41120)
  MoveL 5055 to (232.49, 37.15, 78.65) mm, rotated rx -180 ry 0 rz 180 deg; joints [-156.239, -72.816, -47.89, 40.767, 38.101, -34.155]
  MoveL 5056 to (232.49, 37.15, 78.65) mm, rotated rx -180 ry 0 rz 180 deg; joints [-156.239, -72.816, -47.89, 40.767, 38.101, -34.155]
  Call Extruder(201.56919)
  MoveL 5057 to (232.74, 37.26, 78.65) mm, rotated rx -180 ry 0 rz 180 deg; joints [-156.239, -72.851, -47.813, 40.801, 38.07, -34.199]
  MoveL 5058 to (232.74, 37.26, 78.65) mm, rotated rx -180 ry 0 rz 180 deg; joints [-156.239, -72.851, -47.813, 40.801, 38.07, -34.199]
  Call Extruder(201.72780)
  MoveL 5059 to (232.99, 37.36, 78.65) mm, rotated rx -180 ry 0 rz -180 deg; joints [-156.239, -72.887, -47.736, 40.835, 38.039, -34.242]
  MoveL 5060 to (232.99, 37.36, 78.65) mm, rotated rx -180 ry 0 rz -180 deg; joints [-156.239, -72.887, -47.736, 40.835, 38.039, -34.242]
  Call Extruder(201.93396)
  MoveL 5061 to (233.29, 37.54, 78.65) mm, rotated rx 180 ry 0 rz 180 deg; joints [-156.236, -72.933, -47.637, 40.884, 38.001, -34.302]
  MoveL 5062 to (233.29, 37.54, 78.65) mm, rotated rx 180 ry 0 rz 180 deg; joints [-156.236, -72.933, -47.637, 40.884, 38.001, -34.302]
  Call Extruder(202.14091)
  MoveL 5063 to (233.6, 37.71, 78.65) mm, rotated rx 180 ry 0 rz -180 deg; joints [-156.232, -72.979, -47.538, 40.934, 37.963, -34.363]
  MoveL 5064 to (233.6, 37.71, 78.65) mm, rotated rx 180 ry 0 rz -180 deg; joints [-156.232, -72.979, -47.538, 40.934, 37.963, -34.363]
  Call Extruder(202.34863)
  MoveL 5065 to (233.9, 37.89, 78.65) mm, rotated rx -180 ry 0 rz 180 deg; joints [-156.228, -73.025, -47.438, 40.984, 37.925, -34.424]
  MoveL 5066 to (233.9, 37.89, 78.65) mm, rotated rx -180 ry 0 rz 180 deg; joints [-156.228, -73.025, -47.438, 40.984, 37.925, -34.424]
  Call Extruder(202.55713)
  MoveL 5067 to (234.21, 38.06, 78.65) mm, rotated rx -180 ry 0 rz 180 deg; joints [-156.224, -73.072, -47.338, 41.034, 37.886, -34.485]
  MoveL 5068 to (234.21, 38.06, 78.65) mm, rotated rx -180 ry 0 rz 180 deg; joints [-156.224, -73.072, -47.338, 41.034, 37.886, -34.485]
  Call Extruder(202.73668)
  MoveL 5069 to (234.45, 38.24, 78.65) mm, rotated rx 180 ry 0 rz 180 deg; joints [-156.218, -73.111, -47.254, 41.08, 37.856, -34.539]
  MoveL 5070 to (234.45, 38.24, 78.65) mm, rotated rx 180 ry 0 rz 180 deg; joints [-156.218, -73.111, -47.254, 41.08, 37.856, -34.539]
  Call Extruder(203.07009)
  MoveL 5071 to (234.9, 38.57, 78.65) mm, rotated rx 180 ry 0 rz 180 deg; joints [-156.206, -73.184, -47.098, 41.167, 37.8, -34.641]
  MoveL 5072 to (234.9, 38.57, 78.65) mm, rotated rx 180 ry 0 rz 180 deg; joints [-156.206, -73.184, -47.098, 41.167, 37.8, -34.641]
  Call Extruder(203.40469)
  MoveL 5073 to (235.35, 38.9, 78.65) mm, rotated rx -180 ry 0 rz 180 deg; joints [-156.195, -73.257, -46.941, 41.253, 37.743, -34.744]
  Call Extruder(204.23264)
  MoveL 5074 to (236.39, 39.81, 78.65) mm, rotated rx 180 ry 0 rz 180 deg; joints [-156.154, -73.434, -46.562, 41.482, 37.615, -35.006]
  Call Extruder(205.06059)
  MoveL 5075 to (237.3, 40.85, 78.65) mm, rotated rx -180 ry 0 rz -180 deg; joints [-156.097, -73.603, -46.198, 41.726, 37.503, -35.278]
  Call Extruder(205.22789)
  MoveL 5076 to (237.47, 41.07, 78.65) mm, rotated rx 180 ry 0 rz 180 deg; joints [-156.083, -73.636, -46.128, 41.777, 37.483, -35.334]
  MoveL 5077 to (237.47, 41.07, 78.65) mm, rotated rx 180 ry 0 rz 180 deg; joints [-156.083, -73.636, -46.128, 41.777, 37.483, -35.334]
  Call Extruder(205.56130)
  MoveL 5078 to (237.8, 41.52, 78.65) mm, rotated rx -180 ry 0 rz 180 deg; joints [-156.055, -73.702, -45.987, 41.879, 37.443, -35.445]
  MoveL 5079 to (237.8, 41.52, 78.65) mm, rotated rx -180 ry 0 rz 180 deg; joints [-156.055, -73.702, -45.987, 41.879, 37.443, -35.445]
  Call Extruder(205.89353)
  MoveL 5080 to (238.12, 41.98, 78.65) mm, rotated rx 180 ry 0 rz -180 deg; joints [-156.028, -73.768, -45.846, 41.982, 37.403, -35.557]
  MoveL 5081 to (238.12, 41.98, 78.65) mm, rotated rx 180 ry 0 rz -180 deg; joints [-156.028, -73.768, -45.846, 41.982, 37.403, -35.557]
  Call Extruder(206.01123)
  MoveL 5082 to (238.22, 42.15, 78.65) mm, rotated rx 180 ry 0 rz 180 deg; joints [-156.016, -73.79, -45.799, 42.019, 37.391, -35.597]
  MoveL 5083 to (238.22, 42.15, 78.65) mm, rotated rx 180 ry 0 rz 180 deg; joints [-156.016, -73.79, -45.799, 42.019, 37.391, -35.597]
  Call Extruder(206.21895)
  MoveL 5084 to (238.4, 42.45, 78.65) mm, rotated rx 180 ry 0 rz -180 deg; joints [-155.996, -73.829, -45.716, 42.085, 37.37, -35.668]
  MoveL 5085 to (238.4, 42.45, 78.65) mm, rotated rx 180 ry 0 rz -180 deg; joints [-155.996, -73.829, -45.716, 42.085, 37.37, -35.668]
  Call Extruder(206.42590)
  MoveL 5086 to (238.57, 42.75, 78.65) mm, rotated rx -180 ry 0 rz 180 deg; joints [-155.976, -73.868, -45.633, 42.151, 37.349, -35.738]
  MoveL 5087 to (238.57, 42.75, 78.65) mm, rotated rx -180 ry 0 rz 180 deg; joints [-155.976, -73.868, -45.633, 42.151, 37.349, -35.738]
  Call Extruder(206.63206)
  MoveL 5088 to (238.75, 43.06, 78.65) mm, rotated rx -180 ry 0 rz 180 deg; joints [-155.956, -73.907, -45.549, 42.217, 37.328, -35.809]
  MoveL 5089 to (238.75, 43.06, 78.65) mm, rotated rx -180 ry 0 rz 180 deg; joints [-155.956, -73.907, -45.549, 42.217, 37.328, -35.809]
  Call Extruder(206.81375)
  MoveL 5090 to (238.89, 43.34, 78.65) mm, rotated rx 180 ry 0 rz 180 deg; joints [-155.937, -73.94, -45.478, 42.276, 37.311, -35.871]
  MoveL 5091 to (238.89, 43.34, 78.65) mm, rotated rx 180 ry 0 rz 180 deg; joints [-155.937, -73.94, -45.478, 42.276, 37.311, -35.871]
  Call Extruder(206.97176)
  MoveL 5092 to (239, 43.58, 78.65) mm, rotated rx -180 ry 0 rz -180 deg; joints [-155.919, -73.967, -45.419, 42.327, 37.298, -35.925]
  MoveL 5093 to (239, 43.58, 78.65) mm, rotated rx -180 ry 0 rz -180 deg; joints [-155.919, -73.967, -45.419, 42.327, 37.298, -35.925]
  Call Extruder(207.12917)
  MoveL 5094 to (239.1, 43.83, 78.65) mm, rotated rx -180 ry 0 rz -180 deg; joints [-155.901, -73.995, -45.361, 42.379, 37.286, -35.979]
  MoveL 5095 to (239.1, 43.83, 78.65) mm, rotated rx -180 ry 0 rz -180 deg; joints [-155.901, -73.995, -45.361, 42.379, 37.286, -35.979]
  Call Extruder(207.31188)
  MoveL 5096 to (239.23, 44.12, 78.65) mm, rotated rx 180 ry 0 rz 180 deg; joints [-155.879, -74.026, -45.293, 42.439, 37.272, -36.041]
  MoveL 5097 to (239.23, 44.12, 78.65) mm, rotated rx 180 ry 0 rz 180 deg; joints [-155.879, -74.026, -45.293, 42.439, 37.272, -36.041]
  Call Extruder(207.49384)
  MoveL 5098 to (239.35, 44.42, 78.65) mm, rotated rx 180 ry 0 rz -180 deg; joints [-155.858, -74.058, -45.225, 42.5, 37.258, -36.104]
  MoveL 5099 to (239.35, 44.42, 78.65) mm, rotated rx 180 ry 0 rz -180 deg; joints [-155.858, -74.058, -45.225, 42.5, 37.258, -36.104]
  Call Extruder(207.64117)
  MoveL 5100 to (239.44, 44.66, 78.65) mm, rotated rx 180 ry 0 rz -180 deg; joints [-155.84, -74.083, -45.172, 42.549, 37.247, -36.155]
  MoveL 5101 to (239.44, 44.66, 78.65) mm, rotated rx 180 ry 0 rz -180 deg; joints [-155.84, -74.083, -45.172, 42.549, 37.247, -36.155]
  Call Extruder(207.75441)
  MoveL 5102 to (239.5, 44.85, 78.65) mm, rotated rx 180 ry 0 rz 180 deg; joints [-155.826, -74.102, -45.132, 42.587, 37.24, -36.194]
  MoveL 5103 to (239.5, 44.85, 78.65) mm, rotated rx 180 ry 0 rz 180 deg; joints [-155.826, -74.102, -45.132, 42.587, 37.24, -36.194]
  Call Extruder(207.86720)
  MoveL 5104 to (239.56, 45.03, 78.65) mm, rotated rx -180 ry 0 rz 180 deg; joints [-155.811, -74.12, -45.093, 42.624, 37.233, -36.232]
  MoveL 5105 to (239.56, 45.03, 78.65) mm, rotated rx -180 ry 0 rz 180 deg; joints [-155.811, -74.12, -45.093, 42.624, 37.233, -36.232]
  Call Extruder(207.97954)
  MoveL 5106 to (239.62, 45.22, 78.65) mm, rotated rx -180 ry 0 rz -180 deg; joints [-155.797, -74.139, -45.054, 42.662, 37.226, -36.271]
  MoveL 5107 to (239.62, 45.22, 78.65) mm, rotated rx -180 ry 0 rz -180 deg; joints [-155.797, -74.139, -45.054, 42.662, 37.226, -36.271]
  Call Extruder(208.09145)
  MoveL 5108 to (239.68, 45.41, 78.65) mm, rotated rx 180 ry 0 rz 180 deg; joints [-155.783, -74.157, -45.014, 42.7, 37.219, -36.309]
  MoveL 5109 to (239.68, 45.41, 78.65) mm, rotated rx 180 ry 0 rz 180 deg; joints [-155.783, -74.157, -45.014, 42.7, 37.219, -36.309]
  Call Extruder(208.21285)
  MoveL 5110 to (239.75, 45.62, 78.65) mm, rotated rx -180 ry 0 rz 180 deg; joints [-155.767, -74.177, -44.972, 42.741, 37.212, -36.352]
  MoveL 5111 to (239.75, 45.62, 78.65) mm, rotated rx -180 ry 0 rz 180 deg; joints [-155.767, -74.177, -44.972, 42.741, 37.212, -36.352]
  Call Extruder(208.34364)
  MoveL 5112 to (239.81, 45.84, 78.65) mm, rotated rx 180 ry 0 rz 180 deg; joints [-155.75, -74.199, -44.926, 42.786, 37.205, -36.397]
  MoveL 5113 to (239.81, 45.84, 78.65) mm, rotated rx 180 ry 0 rz 180 deg; joints [-155.75, -74.199, -44.926, 42.786, 37.205, -36.397]
  Call Extruder(208.47386)
  MoveL 5114 to (239.88, 46.06, 78.65) mm, rotated rx 180 ry 0 rz 180 deg; joints [-155.733, -74.22, -44.881, 42.83, 37.197, -36.442]
  MoveL 5115 to (239.88, 46.06, 78.65) mm, rotated rx 180 ry 0 rz 180 deg; joints [-155.733, -74.22, -44.881, 42.83, 37.197, -36.442]
  Call Extruder(208.60352)
  MoveL 5116 to (239.95, 46.29, 78.65) mm, rotated rx 180 ry 0 rz 180 deg; joints [-155.715, -74.241, -44.835, 42.875, 37.19, -36.488]
  MoveL 5117 to (239.95, 46.29, 78.65) mm, rotated rx 180 ry 0 rz 180 deg; joints [-155.715, -74.241, -44.835, 42.875, 37.19, -36.488]
  Call Extruder(208.73262)
  MoveL 5118 to (240.02, 46.51, 78.65) mm, rotated rx 180 ry 0 rz 180 deg; joints [-155.698, -74.263, -44.789, 42.92, 37.182, -36.533]
  MoveL 5119 to (240.02, 46.51, 78.65) mm, rotated rx 180 ry 0 rz 180 deg; joints [-155.698, -74.263, -44.789, 42.92, 37.182, -36.533]
  Call Extruder(208.84768)
  MoveL 5120 to (240.06, 46.72, 78.65) mm, rotated rx -180 ry 0 rz -180 deg; joints [-155.682, -74.28, -44.752, 42.959, 37.177, -36.573]
  MoveL 5121 to (240.06, 46.72, 78.65) mm, rotated rx -180 ry 0 rz -180 deg; joints [-155.682, -74.28, -44.752, 42.959, 37.177, -36.573]
  Call Extruder(208.96228)
  MoveL 5122 to (240.11, 46.92, 78.65) mm, rotated rx 180 ry 0 rz 180 deg; joints [-155.665, -74.298, -44.715, 42.999, 37.173, -36.613]
  MoveL 5123 to (240.11, 46.92, 78.65) mm, rotated rx 180 ry 0 rz 180 deg; joints [-155.665, -74.298, -44.715, 42.999, 37.173, -36.613]
  Call Extruder(209.07643)
  MoveL 5124 to (240.15, 47.12, 78.65) mm, rotated rx 180 ry 0 rz 180 deg; joints [-155.649, -74.315, -44.678, 43.038, 37.168, -36.652]
  MoveL 5125 to (240.15, 47.12, 78.65) mm, rotated rx 180 ry 0 rz 180 deg; joints [-155.649, -74.315, -44.678, 43.038, 37.168, -36.652]
  Call Extruder(209.19012)
  MoveL 5126 to (240.2, 47.33, 78.65) mm, rotated rx 180 ry 0 rz 180 deg; joints [-155.633, -74.332, -44.64, 43.078, 37.163, -36.692]
  MoveL 5127 to (240.2, 47.33, 78.65) mm, rotated rx 180 ry 0 rz 180 deg; joints [-155.633, -74.332, -44.64, 43.078, 37.163, -36.692]
  Call Extruder(209.31554)
  MoveL 5128 to (240.24, 47.55, 78.65) mm, rotated rx 180 ry 0 rz 180 deg; joints [-155.614, -74.351, -44.6, 43.121, 37.158, -36.736]
  MoveL 5129 to (240.24, 47.55, 78.65) mm, rotated rx 180 ry 0 rz 180 deg; joints [-155.614, -74.351, -44.6, 43.121, 37.158, -36.736]
  Call Extruder(209.45251)
  MoveL 5130 to (240.29, 47.8, 78.65) mm, rotated rx -180 ry 0 rz 180 deg; joints [-155.594, -74.372, -44.556, 43.169, 37.153, -36.783]
  MoveL 5131 to (240.29, 47.8, 78.65) mm, rotated rx -180 ry 0 rz 180 deg; joints [-155.594, -74.372, -44.556, 43.169, 37.153, -36.783]
  Call Extruder(209.58888)
  MoveL 5132 to (240.34, 48.05, 78.65) mm, rotated rx -180 ry 0 rz 180 deg; joints [-155.574, -74.393, -44.511, 43.217, 37.148, -36.831]
  MoveL 5133 to (240.34, 48.05, 78.65) mm, rotated rx -180 ry 0 rz 180 deg; joints [-155.574, -74.393, -44.511, 43.217, 37.148, -36.831]
  Call Extruder(209.72464)
  MoveL 5134 to (240.39, 48.3, 78.65) mm, rotated rx -180 ry 0 rz 180 deg; joints [-155.554, -74.414, -44.467, 43.265, 37.143, -36.879]
  MoveL 5135 to (240.39, 48.3, 78.65) mm, rotated rx -180 ry 0 rz 180 deg; joints [-155.554, -74.414, -44.467, 43.265, 37.143, -36.879]
  Call Extruder(209.85978)
  MoveL 5136 to (240.44, 48.55, 78.65) mm, rotated rx 180 ry 0 rz 180 deg; joints [-155.534, -74.435, -44.423, 43.313, 37.138, -36.927]
  MoveL 5137 to (240.44, 48.55, 78.65) mm, rotated rx 180 ry 0 rz 180 deg; joints [-155.534, -74.435, -44.423, 43.313, 37.138, -36.927]
  Call Extruder(209.99432)
  MoveL 5138 to (240.49, 48.8, 78.65) mm, rotated rx -180 ry 0 rz 180 deg; joints [-155.514, -74.455, -44.378, 43.361, 37.133, -36.975]
  MoveL 5139 to (240.49, 48.8, 78.65) mm, rotated rx -180 ry 0 rz 180 deg; joints [-155.514, -74.455, -44.378, 43.361, 37.133, -36.975]
  Call Extruder(210.12825)
  MoveL 5140 to (240.54, 49.05, 78.65) mm, rotated rx -180 ry 0 rz 180 deg; joints [-155.494, -74.476, -44.334, 43.409, 37.128, -37.023]
  MoveL 5141 to (240.54, 49.05, 78.65) mm, rotated rx -180 ry 0 rz 180 deg; joints [-155.494, -74.476, -44.334, 43.409, 37.128, -37.023]
  Call Extruder(210.27611)
  MoveL 5142 to (240.59, 49.33, 78.65) mm, rotated rx -180 ry 0 rz -180 deg; joints [-155.471, -74.499, -44.286, 43.462, 37.123, -37.076]
  MoveL 5143 to (240.59, 49.33, 78.65) mm, rotated rx -180 ry 0 rz -180 deg; joints [-155.471, -74.499, -44.286, 43.462, 37.123, -37.076]
  Call Extruder(210.43786)
  MoveL 5144 to (240.64, 49.63, 78.65) mm, rotated rx 180 ry 0 rz -180 deg; joints [-155.446, -74.523, -44.235, 43.52, 37.119, -37.133]
  MoveL 5145 to (240.64, 49.63, 78.65) mm, rotated rx 180 ry 0 rz -180 deg; joints [-155.446, -74.523, -44.235, 43.52, 37.119, -37.133]
  Call Extruder(210.59887)
  MoveL 5146 to (240.69, 49.94, 78.65) mm, rotated rx 180 ry 0 rz -180 deg; joints [-155.421, -74.547, -44.183, 43.578, 37.114, -37.191]
  MoveL 5147 to (240.69, 49.94, 78.65) mm, rotated rx 180 ry 0 rz -180 deg; joints [-155.421, -74.547, -44.183, 43.578, 37.114, -37.191]
  Call Extruder(210.75916)
  MoveL 5148 to (240.74, 50.24, 78.65) mm, rotated rx 180 ry 0 rz 180 deg; joints [-155.396, -74.571, -44.132, 43.635, 37.11, -37.248]
  MoveL 5149 to (240.74, 50.24, 78.65) mm, rotated rx 180 ry 0 rz 180 deg; joints [-155.396, -74.571, -44.132, 43.635, 37.11, -37.248]
  Call Extruder(210.91872)
  MoveL 5150 to (240.78, 50.55, 78.65) mm, rotated rx -180 ry 0 rz 180 deg; joints [-155.371, -74.595, -44.08, 43.694, 37.105, -37.306]
  MoveL 5151 to (240.78, 50.55, 78.65) mm, rotated rx -180 ry 0 rz 180 deg; joints [-155.371, -74.595, -44.08, 43.694, 37.105, -37.306]
  Call Extruder(211.07756)
  MoveL 5152 to (240.83, 50.86, 78.65) mm, rotated rx 180 ry 0 rz 180 deg; joints [-155.346, -74.62, -44.029, 43.752, 37.1, -37.364]
  MoveL 5153 to (240.83, 50.86, 78.65) mm, rotated rx 180 ry 0 rz 180 deg; joints [-155.346, -74.62, -44.029, 43.752, 37.1, -37.364]
  Call Extruder(211.25623)
  MoveL 5154 to (240.88, 51.2, 78.65) mm, rotated rx -180 ry 0 rz -180 deg; joints [-155.317, -74.646, -43.972, 43.817, 37.096, -37.428]
  MoveL 5155 to (240.88, 51.2, 78.65) mm, rotated rx -180 ry 0 rz -180 deg; joints [-155.317, -74.646, -43.972, 43.817, 37.096, -37.428]
  Call Extruder(211.45467)
  MoveL 5156 to (240.92, 51.59, 78.65) mm, rotated rx -180 ry 0 rz -180 deg; joints [-155.285, -74.675, -43.911, 43.889, 37.092, -37.5]
  MoveL 5157 to (240.92, 51.59, 78.65) mm, rotated rx -180 ry 0 rz -180 deg; joints [-155.285, -74.675, -43.911, 43.889, 37.092, -37.5]
  Call Extruder(211.65225)
  MoveL 5158 to (240.97, 51.98, 78.65) mm, rotated rx 180 ry 0 rz 180 deg; joints [-155.252, -74.704, -43.849, 43.962, 37.089, -37.571]
  MoveL 5159 to (240.97, 51.98, 78.65) mm, rotated rx 180 ry 0 rz 180 deg; joints [-155.252, -74.704, -43.849, 43.962, 37.089, -37.571]
  Call Extruder(211.84895)
  MoveL 5160 to (241.02, 52.36, 78.65) mm, rotated rx 180 ry 0 rz 180 deg; joints [-155.22, -74.733, -43.787, 44.034, 37.085, -37.643]
  MoveL 5161 to (241.02, 52.36, 78.65) mm, rotated rx 180 ry 0 rz 180 deg; joints [-155.22, -74.733, -43.787, 44.034, 37.085, -37.643]
  Call Extruder(212.04479)
  MoveL 5162 to (241.06, 52.75, 78.65) mm, rotated rx -180 ry 0 rz 180 deg; joints [-155.188, -74.762, -43.726, 44.106, 37.081, -37.714]
  MoveL 5163 to (241.06, 52.75, 78.65) mm, rotated rx -180 ry 0 rz 180 deg; joints [-155.188, -74.762, -43.726, 44.106, 37.081, -37.714]
  Call Extruder(212.34023)
  MoveL 5164 to (241.11, 53.34, 78.65) mm, rotated rx 180 ry 0 rz 180 deg; joints [-155.138, -74.804, -43.638, 44.215, 37.078, -37.82]
  MoveL 5165 to (241.11, 53.34, 78.65) mm, rotated rx 180 ry 0 rz 180 deg; joints [-155.138, -74.804, -43.638, 44.215, 37.078, -37.82]
  Call Extruder(212.63433)
  MoveL 5166 to (241.16, 53.93, 78.65) mm, rotated rx -180 ry 0 rz 180 deg; joints [-155.088, -74.845, -43.55, 44.323, 37.076, -37.926]
  MoveL 5167 to (241.16, 53.93, 78.65) mm, rotated rx -180 ry 0 rz 180 deg; joints [-155.088, -74.845, -43.55, 44.323, 37.076, -37.926]
  Call Extruder(212.92711)
  MoveL 5168 to (241.2, 54.52, 78.65) mm, rotated rx 180 ry 0 rz -180 deg; joints [-155.038, -74.887, -43.462, 44.432, 37.073, -38.033]
  MoveL 5169 to (241.2, 54.52, 78.65) mm, rotated rx 180 ry 0 rz -180 deg; joints [-155.038, -74.887, -43.462, 44.432, 37.073, -38.033]
  Call Extruder(213.50056)
  MoveL 5170 to (241.25, 55.68, 78.65) mm, rotated rx 180 ry 0 rz -180 deg; joints [-154.938, -74.963, -43.299, 44.642, 37.074, -38.237]
  MoveL 5171 to (241.25, 55.68, 78.65) mm, rotated rx 180 ry 0 rz -180 deg; joints [-154.938, -74.963, -43.299, 44.642, 37.074, -38.237]
  Call Extruder(214.21439)
  MoveL 5172 to (241.29, 57.14, 78.65) mm, rotated rx 180 ry 0 rz 180 deg; joints [-154.812, -75.057, -43.1, 44.904, 37.077, -38.49]
  Call Extruder(256.27928)
  MoveL 5173 to (241.29, 142.86, 78.65) mm, rotated rx -180 ry 0 rz 180 deg; joints [-147.778, -81.977, -28.713, 60.726, 37.681, -54.69]
  Call Extruder(256.70771)
  MoveL 5174 to (241.27, 143.73, 78.65) mm, rotated rx -180 ry 0 rz 180 deg; joints [-147.711, -82.068, -28.529, 60.896, 37.69, -54.874]
  MoveL 5175 to (241.27, 143.73, 78.65) mm, rotated rx -180 ry 0 rz 180 deg; joints [-147.711, -82.068, -28.529, 60.896, 37.69, -54.874]
  Call Extruder(257.28116)
  MoveL 5176 to (241.22, 144.9, 78.65) mm, rotated rx 180 ry 0 rz -180 deg; joints [-147.62, -82.185, -28.289, 61.119, 37.706, -55.116]
  MoveL 5177 to (241.22, 144.9, 78.65) mm, rotated rx 180 ry 0 rz -180 deg; joints [-147.62, -82.185, -28.289, 61.119, 37.706, -55.116]
  Call Extruder(257.71549)
  MoveL 5178 to (241.18, 145.77, 78.65) mm, rotated rx 180 ry 0 rz 180 deg; joints [-147.551, -82.272, -28.112, 61.286, 37.719, -55.296]
  MoveL 5179 to (241.18, 145.77, 78.65) mm, rotated rx 180 ry 0 rz 180 deg; joints [-147.551, -82.272, -28.112, 61.286, 37.719, -55.296]
  Call Extruder(258.00960)
  MoveL 5180 to (241.13, 146.36, 78.65) mm, rotated rx 180 ry 0 rz -180 deg; joints [-147.504, -82.328, -27.998, 61.396, 37.73, -55.414]
  MoveL 5181 to (241.13, 146.36, 78.65) mm, rotated rx 180 ry 0 rz -180 deg; joints [-147.504, -82.328, -27.998, 61.396, 37.73, -55.414]
  Call Extruder(258.30504)
  MoveL 5182 to (241.09, 146.95, 78.65) mm, rotated rx -180 ry 0 rz 180 deg; joints [-147.457, -82.384, -27.883, 61.506, 37.74, -55.533]
  MoveL 5183 to (241.09, 146.95, 78.65) mm, rotated rx -180 ry 0 rz 180 deg; joints [-147.457, -82.384, -27.883, 61.506, 37.74, -55.533]
  Call Extruder(258.55130)
  MoveL 5184 to (241.04, 147.44, 78.65) mm, rotated rx 180 ry 0 rz 180 deg; joints [-147.417, -82.43, -27.79, 61.596, 37.75, -55.63]
  MoveL 5185 to (241.04, 147.44, 78.65) mm, rotated rx 180 ry 0 rz 180 deg; joints [-147.417, -82.43, -27.79, 61.596, 37.75, -55.63]
  Call Extruder(258.74800)
  MoveL 5186 to (240.99, 147.83, 78.65) mm, rotated rx -180 ry 0 rz -180 deg; joints [-147.386, -82.465, -27.719, 61.666, 37.759, -55.705]
  MoveL 5187 to (240.99, 147.83, 78.65) mm, rotated rx -180 ry 0 rz -180 deg; joints [-147.386, -82.465, -27.719, 61.666, 37.759, -55.705]
  Call Extruder(258.94558)
  MoveL 5188 to (240.95, 148.22, 78.65) mm, rotated rx 180 ry 0 rz 180 deg; joints [-147.354, -82.5, -27.648, 61.736, 37.768, -55.78]
  MoveL 5189 to (240.95, 148.22, 78.65) mm, rotated rx 180 ry 0 rz 180 deg; joints [-147.354, -82.5, -27.648, 61.736, 37.768, -55.78]
  Call Extruder(259.14402)
  MoveL 5190 to (240.9, 148.6, 78.65) mm, rotated rx 180 ry 0 rz -180 deg; joints [-147.322, -82.535, -27.577, 61.806, 37.777, -55.855]
  MoveL 5191 to (240.9, 148.6, 78.65) mm, rotated rx 180 ry 0 rz -180 deg; joints [-147.322, -82.535, -27.577, 61.806, 37.777, -55.855]
  Call Extruder(259.34333)
  MoveL 5192 to (240.86, 148.99, 78.65) mm, rotated rx -180 ry 0 rz 180 deg; joints [-147.291, -82.57, -27.506, 61.876, 37.786, -55.93]
  MoveL 5193 to (240.86, 148.99, 78.65) mm, rotated rx -180 ry 0 rz 180 deg; joints [-147.291, -82.57, -27.506, 61.876, 37.786, -55.93]
  Call Extruder(259.50216)
  MoveL 5194 to (240.81, 149.3, 78.65) mm, rotated rx -180 ry 0 rz 180 deg; joints [-147.265, -82.595, -27.453, 61.93, 37.795, -55.986]
  MoveL 5195 to (240.81, 149.3, 78.65) mm, rotated rx -180 ry 0 rz 180 deg; joints [-147.265, -82.595, -27.453, 61.93, 37.795, -55.986]
  Call Extruder(259.66172)
  MoveL 5196 to (240.76, 149.6, 78.65) mm, rotated rx -180 ry 0 rz -180 deg; joints [-147.24, -82.621, -27.401, 61.983, 37.804, -56.043]
  MoveL 5197 to (240.76, 149.6, 78.65) mm, rotated rx -180 ry 0 rz -180 deg; joints [-147.24, -82.621, -27.401, 61.983, 37.804, -56.043]
  Call Extruder(259.82201)
  MoveL 5198 to (240.71, 149.91, 78.65) mm, rotated rx 180 ry 0 rz 180 deg; joints [-147.214, -82.647, -27.349, 62.037, 37.812, -56.1]
  MoveL 5199 to (240.71, 149.91, 78.65) mm, rotated rx 180 ry 0 rz 180 deg; joints [-147.214, -82.647, -27.349, 62.037, 37.812, -56.1]
  Call Extruder(259.98302)
  MoveL 5200 to (240.66, 150.21, 78.65) mm, rotated rx -180 ry 0 rz 180 deg; joints [-147.189, -82.672, -27.296, 62.09, 37.821, -56.156]
  MoveL 5201 to (240.66, 150.21, 78.65) mm, rotated rx -180 ry 0 rz 180 deg; joints [-147.189, -82.672, -27.296, 62.09, 37.821, -56.156]
  Call Extruder(260.14477)
  MoveL 5202 to (240.61, 150.52, 78.65) mm, rotated rx 180 ry 0 rz 180 deg; joints [-147.163, -82.698, -27.244, 62.144, 37.83, -56.213]
  MoveL 5203 to (240.61, 150.52, 78.65) mm, rotated rx 180 ry 0 rz 180 deg; joints [-147.163, -82.698, -27.244, 62.144, 37.83, -56.213]
  Call Extruder(260.30724)
  MoveL 5204 to (240.56, 150.83, 78.65) mm, rotated rx -180 ry 0 rz -180 deg; joints [-147.138, -82.724, -27.191, 62.198, 37.838, -56.27]
  MoveL 5205 to (240.56, 150.83, 78.65) mm, rotated rx -180 ry 0 rz -180 deg; joints [-147.138, -82.724, -27.191, 62.198, 37.838, -56.27]
  Call Extruder(260.44117)
  MoveL 5206 to (240.52, 151.07, 78.65) mm, rotated rx -180 ry 0 rz 180 deg; joints [-147.117, -82.744, -27.151, 62.24, 37.846, -56.314]
  MoveL 5207 to (240.52, 151.07, 78.65) mm, rotated rx -180 ry 0 rz 180 deg; joints [-147.117, -82.744, -27.151, 62.24, 37.846, -56.314]
  Call Extruder(260.57570)
  MoveL 5208 to (240.47, 151.32, 78.65) mm, rotated rx 180 ry 0 rz 180 deg; joints [-147.095, -82.763, -27.112, 62.282, 37.855, -56.358]
  MoveL 5209 to (240.47, 151.32, 78.65) mm, rotated rx 180 ry 0 rz 180 deg; joints [-147.095, -82.763, -27.112, 62.282, 37.855, -56.358]
  Call Extruder(260.71085)
  MoveL 5210 to (240.42, 151.57, 78.65) mm, rotated rx 180 ry 0 rz 180 deg; joints [-147.074, -82.782, -27.072, 62.324, 37.863, -56.402]
  MoveL 5211 to (240.42, 151.57, 78.65) mm, rotated rx 180 ry 0 rz 180 deg; joints [-147.074, -82.782, -27.072, 62.324, 37.863, -56.402]
  Call Extruder(260.84661)
  MoveL 5212 to (240.37, 151.82, 78.65) mm, rotated rx 180 ry 0 rz -180 deg; joints [-147.053, -82.802, -27.033, 62.366, 37.871, -56.447]
  MoveL 5213 to (240.37, 151.82, 78.65) mm, rotated rx 180 ry 0 rz -180 deg; joints [-147.053, -82.802, -27.033, 62.366, 37.871, -56.447]
  Call Extruder(260.98297)
  MoveL 5214 to (240.32, 152.07, 78.65) mm, rotated rx 180 ry 0 rz 180 deg; joints [-147.032, -82.822, -26.993, 62.408, 37.88, -56.491]
  MoveL 5215 to (240.32, 152.07, 78.65) mm, rotated rx 180 ry 0 rz 180 deg; joints [-147.032, -82.822, -26.993, 62.408, 37.88, -56.491]
  Call Extruder(261.11995)
  MoveL 5216 to (240.27, 152.32, 78.65) mm, rotated rx -180 ry 0 rz 180 deg; joints [-147.011, -82.841, -26.953, 62.45, 37.888, -56.535]
  MoveL 5217 to (240.27, 152.32, 78.65) mm, rotated rx -180 ry 0 rz 180 deg; joints [-147.011, -82.841, -26.953, 62.45, 37.888, -56.535]
  Call Extruder(261.25754)
  MoveL 5218 to (240.22, 152.57, 78.65) mm, rotated rx 180 ry 0 rz 180 deg; joints [-146.989, -82.861, -26.913, 62.492, 37.896, -56.579]
  MoveL 5219 to (240.22, 152.57, 78.65) mm, rotated rx 180 ry 0 rz 180 deg; joints [-146.989, -82.861, -26.913, 62.492, 37.896, -56.579]
  Call Extruder(261.37124)
  MoveL 5220 to (240.17, 152.77, 78.65) mm, rotated rx 180 ry 0 rz 180 deg; joints [-146.972, -82.876, -26.881, 62.526, 37.904, -56.615]
  MoveL 5221 to (240.17, 152.77, 78.65) mm, rotated rx 180 ry 0 rz 180 deg; joints [-146.972, -82.876, -26.881, 62.526, 37.904, -56.615]
  Call Extruder(261.48539)
  MoveL 5222 to (240.13, 152.98, 78.65) mm, rotated rx 180 ry 0 rz -180 deg; joints [-146.954, -82.892, -26.85, 62.56, 37.911, -56.65]
  MoveL 5223 to (240.13, 152.98, 78.65) mm, rotated rx 180 ry 0 rz -180 deg; joints [-146.954, -82.892, -26.85, 62.56, 37.911, -56.65]
  Call Extruder(261.59999)
  MoveL 5224 to (240.08, 153.18, 78.65) mm, rotated rx 180 ry 0 rz 180 deg; joints [-146.937, -82.907, -26.819, 62.594, 37.918, -56.686]
  MoveL 5225 to (240.08, 153.18, 78.65) mm, rotated rx 180 ry 0 rz 180 deg; joints [-146.937, -82.907, -26.819, 62.594, 37.918, -56.686]
  Call Extruder(261.71505)
  MoveL 5226 to (240.04, 153.39, 78.65) mm, rotated rx -180 ry 0 rz -180 deg; joints [-146.919, -82.923, -26.787, 62.628, 37.926, -56.721]
  MoveL 5227 to (240.04, 153.39, 78.65) mm, rotated rx -180 ry 0 rz -180 deg; joints [-146.919, -82.923, -26.787, 62.628, 37.926, -56.721]
  Call Extruder(261.83727)
  MoveL 5228 to (239.98, 153.6, 78.65) mm, rotated rx 180 ry 0 rz 180 deg; joints [-146.9, -82.937, -26.757, 62.662, 37.934, -56.756]
  MoveL 5229 to (239.98, 153.6, 78.65) mm, rotated rx 180 ry 0 rz 180 deg; joints [-146.9, -82.937, -26.757, 62.662, 37.934, -56.756]
  Call Extruder(261.96693)
  MoveL 5230 to (239.92, 153.82, 78.65) mm, rotated rx 180 ry 0 rz 180 deg; joints [-146.88, -82.951, -26.73, 62.696, 37.945, -56.791]
  MoveL 5231 to (239.92, 153.82, 78.65) mm, rotated rx 180 ry 0 rz 180 deg; joints [-146.88, -82.951, -26.73, 62.696, 37.945, -56.791]
  Call Extruder(262.09716)
  MoveL 5232 to (239.85, 154.05, 78.65) mm, rotated rx 180 ry 0 rz -180 deg; joints [-146.86, -82.965, -26.702, 62.73, 37.955, -56.826]
  MoveL 5233 to (239.85, 154.05, 78.65) mm, rotated rx 180 ry 0 rz -180 deg; joints [-146.86, -82.965, -26.702, 62.73, 37.955, -56.826]
  Call Extruder(262.22795)
  MoveL 5234 to (239.78, 154.27, 78.65) mm, rotated rx -180 ry 0 rz -180 deg; joints [-146.84, -82.979, -26.673, 62.764, 37.965, -56.86]
  MoveL 5235 to (239.78, 154.27, 78.65) mm, rotated rx -180 ry 0 rz -180 deg; joints [-146.84, -82.979, -26.673, 62.764, 37.965, -56.86]
  Call Extruder(262.35930)
  MoveL 5236 to (239.71, 154.49, 78.65) mm, rotated rx -180 ry 0 rz 180 deg; joints [-146.82, -82.993, -26.645, 62.799, 37.976, -56.895]
  MoveL 5237 to (239.71, 154.49, 78.65) mm, rotated rx -180 ry 0 rz 180 deg; joints [-146.82, -82.993, -26.645, 62.799, 37.976, -56.895]
  Call Extruder(262.47120)
  MoveL 5238 to (239.65, 154.68, 78.65) mm, rotated rx 180 ry 0 rz 180 deg; joints [-146.803, -83.003, -26.623, 62.827, 37.985, -56.923]
  MoveL 5239 to (239.65, 154.68, 78.65) mm, rotated rx 180 ry 0 rz 180 deg; joints [-146.803, -83.003, -26.623, 62.827, 37.985, -56.923]
  Call Extruder(262.58355)
  MoveL 5240 to (239.59, 154.87, 78.65) mm, rotated rx 180 ry 0 rz 180 deg; joints [-146.785, -83.014, -26.601, 62.855, 37.994, -56.952]
  MoveL 5241 to (239.59, 154.87, 78.65) mm, rotated rx 180 ry 0 rz 180 deg; joints [-146.785, -83.014, -26.601, 62.855, 37.994, -56.952]
  Call Extruder(262.69634)
  MoveL 5242 to (239.53, 155.06, 78.65) mm, rotated rx 180 ry 0 rz 180 deg; joints [-146.768, -83.025, -26.579, 62.883, 38.003, -56.98]
  MoveL 5243 to (239.53, 155.06, 78.65) mm, rotated rx 180 ry 0 rz 180 deg; joints [-146.768, -83.025, -26.579, 62.883, 38.003, -56.98]
  Call Extruder(262.80957)
  MoveL 5244 to (239.47, 155.25, 78.65) mm, rotated rx 180 ry 0 rz 180 deg; joints [-146.751, -83.036, -26.556, 62.911, 38.013, -57.008]
  MoveL 5245 to (239.47, 155.25, 78.65) mm, rotated rx 180 ry 0 rz 180 deg; joints [-146.751, -83.036, -26.556, 62.911, 38.013, -57.008]
  Call Extruder(262.92325)
  MoveL 5246 to (239.41, 155.44, 78.65) mm, rotated rx 180 ry 0 rz 180 deg; joints [-146.734, -83.047, -26.534, 62.939, 38.022, -57.037]
  MoveL 5247 to (239.41, 155.44, 78.65) mm, rotated rx 180 ry 0 rz 180 deg; joints [-146.734, -83.047, -26.534, 62.939, 38.022, -57.037]
  Call Extruder(263.10521)
  MoveL 5248 to (239.29, 155.73, 78.65) mm, rotated rx 180 ry 0 rz 180 deg; joints [-146.706, -83.06, -26.509, 62.978, 38.039, -57.075]
  MoveL 5249 to (239.29, 155.73, 78.65) mm, rotated rx 180 ry 0 rz 180 deg; joints [-146.706, -83.06, -26.509, 62.978, 38.039, -57.075]
  Call Extruder(263.28793)
  MoveL 5250 to (239.17, 156.02, 78.65) mm, rotated rx 180 ry 0 rz 180 deg; joints [-146.678, -83.072, -26.483, 63.017, 38.057, -57.113]
  MoveL 5251 to (239.17, 156.02, 78.65) mm, rotated rx 180 ry 0 rz 180 deg; joints [-146.678, -83.072, -26.483, 63.017, 38.057, -57.113]
  Call Extruder(263.45835)
  MoveL 5252 to (239.05, 156.29, 78.65) mm, rotated rx 180 ry 0 rz 180 deg; joints [-146.652, -83.084, -26.461, 63.053, 38.073, -57.147]
  MoveL 5253 to (239.05, 156.29, 78.65) mm, rotated rx 180 ry 0 rz 180 deg; joints [-146.652, -83.084, -26.461, 63.053, 38.073, -57.147]
  Call Extruder(263.61637)
  MoveL 5254 to (238.94, 156.54, 78.65) mm, rotated rx 180 ry 0 rz 180 deg; joints [-146.628, -83.094, -26.44, 63.086, 38.089, -57.179]
  MoveL 5255 to (238.94, 156.54, 78.65) mm, rotated rx 180 ry 0 rz 180 deg; joints [-146.628, -83.094, -26.44, 63.086, 38.089, -57.179]
  Call Extruder(263.77499)
  MoveL 5256 to (238.84, 156.79, 78.65) mm, rotated rx -180 ry 0 rz 180 deg; joints [-146.604, -83.104, -26.419, 63.119, 38.104, -57.211]
  MoveL 5257 to (238.84, 156.79, 78.65) mm, rotated rx -180 ry 0 rz 180 deg; joints [-146.604, -83.104, -26.419, 63.119, 38.104, -57.211]
  Call Extruder(264.00155)
  MoveL 5258 to (238.65, 157.13, 78.65) mm, rotated rx 180 ry 0 rz -180 deg; joints [-146.57, -83.11, -26.408, 63.156, 38.131, -57.243]
  MoveL 5259 to (238.65, 157.13, 78.65) mm, rotated rx 180 ry 0 rz -180 deg; joints [-146.57, -83.11, -26.408, 63.156, 38.131, -57.243]
  Call Extruder(264.22896)
  MoveL 5260 to (238.46, 157.46, 78.65) mm, rotated rx 180 ry 0 rz -180 deg; joints [-146.536, -83.116, -26.396, 63.193, 38.157, -57.276]
  MoveL 5261 to (238.46, 157.46, 78.65) mm, rotated rx 180 ry 0 rz -180 deg; joints [-146.536, -83.116, -26.396, 63.193, 38.157, -57.276]
  Call Extruder(264.41617)
  MoveL 5262 to (238.3, 157.73, 78.65) mm, rotated rx 180 ry 0 rz 180 deg; joints [-146.507, -83.119, -26.39, 63.222, 38.179, -57.3]
  MoveL 5263 to (238.3, 157.73, 78.65) mm, rotated rx 180 ry 0 rz 180 deg; joints [-146.507, -83.119, -26.39, 63.222, 38.179, -57.3]
  Call Extruder(264.60408)
  MoveL 5264 to (238.13, 158.01, 78.65) mm, rotated rx 180 ry 0 rz -180 deg; joints [-146.479, -83.122, -26.383, 63.25, 38.202, -57.324]
  MoveL 5265 to (238.13, 158.01, 78.65) mm, rotated rx 180 ry 0 rz -180 deg; joints [-146.479, -83.122, -26.383, 63.25, 38.202, -57.324]
  Call Extruder(264.78361)
  MoveL 5266 to (237.96, 158.25, 78.65) mm, rotated rx 180 ry 0 rz 180 deg; joints [-146.452, -83.119, -26.388, 63.271, 38.225, -57.339]
  MoveL 5267 to (237.96, 158.25, 78.65) mm, rotated rx 180 ry 0 rz 180 deg; joints [-146.452, -83.119, -26.388, 63.271, 38.225, -57.339]
  Call Extruder(265.11703)
  MoveL 5268 to (237.63, 158.7, 78.65) mm, rotated rx -180 ry 0 rz 180 deg; joints [-146.402, -83.114, -26.398, 63.308, 38.27, -57.365]
  MoveL 5269 to (237.63, 158.7, 78.65) mm, rotated rx -180 ry 0 rz 180 deg; joints [-146.402, -83.114, -26.398, 63.308, 38.27, -57.365]
  Call Extruder(265.45163)
  MoveL 5270 to (237.3, 159.15, 78.65) mm, rotated rx 180 ry 0 rz 180 deg; joints [-146.352, -83.109, -26.408, 63.346, 38.314, -57.392]
  Call Extruder(266.27957)
  MoveL 5271 to (236.39, 160.19, 78.65) mm, rotated rx 180 ry 0 rz 180 deg; joints [-146.229, -83.071, -26.487, 63.408, 38.436, -57.418]
  Call Extruder(267.10752)
  MoveL 5272 to (235.35, 161.1, 78.65) mm, rotated rx 180 ry 0 rz 180 deg; joints [-146.109, -82.996, -26.638, 63.425, 38.571, -57.389]
  Call Extruder(267.27483)
  MoveL 5273 to (235.13, 161.27, 78.65) mm, rotated rx -180 ry 0 rz -180 deg; joints [-146.086, -82.976, -26.679, 63.422, 38.6, -57.375]
  MoveL 5274 to (235.13, 161.27, 78.65) mm, rotated rx -180 ry 0 rz -180 deg; joints [-146.086, -82.976, -26.679, 63.422, 38.6, -57.375]
  Call Extruder(267.60825)
  MoveL 5275 to (234.68, 161.59, 78.65) mm, rotated rx -180 ry 0 rz 180 deg; joints [-146.039, -82.936, -26.761, 63.416, 38.658, -57.347]
  MoveL 5276 to (234.68, 161.59, 78.65) mm, rotated rx -180 ry 0 rz 180 deg; joints [-146.039, -82.936, -26.761, 63.416, 38.658, -57.347]
  Call Extruder(267.94049)
  MoveL 5277 to (234.22, 161.92, 78.65) mm, rotated rx -180 ry 0 rz 180 deg; joints [-145.992, -82.896, -26.842, 63.411, 38.716, -57.32]
  MoveL 5278 to (234.22, 161.92, 78.65) mm, rotated rx -180 ry 0 rz 180 deg; joints [-145.992, -82.896, -26.842, 63.411, 38.716, -57.32]
  Call Extruder(268.05815)
  MoveL 5279 to (234.05, 162.02, 78.65) mm, rotated rx -180 ry 0 rz -180 deg; joints [-145.976, -82.878, -26.879, 63.404, 38.738, -57.304]
  MoveL 5280 to (234.05, 162.02, 78.65) mm, rotated rx -180 ry 0 rz -180 deg; joints [-145.976, -82.878, -26.879, 63.404, 38.738, -57.304]
  Call Extruder(268.26588)
  MoveL 5281 to (233.75, 162.2, 78.65) mm, rotated rx 180 ry 0 rz 180 deg; joints [-145.947, -82.846, -26.944, 63.392, 38.777, -57.276]
  MoveL 5282 to (233.75, 162.2, 78.65) mm, rotated rx 180 ry 0 rz 180 deg; joints [-145.947, -82.846, -26.944, 63.392, 38.777, -57.276]
  Call Extruder(268.47282)
  MoveL 5283 to (233.45, 162.37, 78.65) mm, rotated rx -180 ry 0 rz 180 deg; joints [-145.919, -82.814, -27.009, 63.379, 38.815, -57.248]
  MoveL 5284 to (233.45, 162.37, 78.65) mm, rotated rx -180 ry 0 rz 180 deg; joints [-145.919, -82.814, -27.009, 63.379, 38.815, -57.248]
  Call Extruder(268.67899)
  MoveL 5285 to (233.14, 162.55, 78.65) mm, rotated rx -180 ry 0 rz 180 deg; joints [-145.891, -82.782, -27.074, 63.367, 38.854, -57.22]
  MoveL 5286 to (233.14, 162.55, 78.65) mm, rotated rx -180 ry 0 rz 180 deg; joints [-145.891, -82.782, -27.074, 63.367, 38.854, -57.22]
  Call Extruder(268.86066)
  MoveL 5287 to (232.87, 162.69, 78.65) mm, rotated rx -180 ry 0 rz 180 deg; joints [-145.866, -82.751, -27.137, 63.352, 38.889, -57.191]
  MoveL 5288 to (232.87, 162.69, 78.65) mm, rotated rx -180 ry 0 rz 180 deg; joints [-145.866, -82.751, -27.137, 63.352, 38.889, -57.191]
  Call Extruder(269.01864)
  MoveL 5289 to (232.62, 162.8, 78.65) mm, rotated rx -180 ry 0 rz -180 deg; joints [-145.845, -82.72, -27.199, 63.335, 38.92, -57.16]
  MoveL 5290 to (232.62, 162.8, 78.65) mm, rotated rx -180 ry 0 rz -180 deg; joints [-145.845, -82.72, -27.199, 63.335, 38.92, -57.16]
  Call Extruder(269.17601)
  MoveL 5291 to (232.37, 162.91, 78.65) mm, rotated rx 180 ry 0 rz 180 deg; joints [-145.825, -82.69, -27.26, 63.319, 38.952, -57.129]
  MoveL 5292 to (232.37, 162.91, 78.65) mm, rotated rx 180 ry 0 rz 180 deg; joints [-145.825, -82.69, -27.26, 63.319, 38.952, -57.129]
  Call Extruder(269.35875)
  MoveL 5293 to (232.08, 163.03, 78.65) mm, rotated rx 180 ry 0 rz 180 deg; joints [-145.801, -82.654, -27.334, 63.298, 38.988, -57.092]
  MoveL 5294 to (232.08, 163.03, 78.65) mm, rotated rx 180 ry 0 rz 180 deg; joints [-145.801, -82.654, -27.334, 63.298, 38.988, -57.092]
  Call Extruder(269.54073)
  MoveL 5295 to (231.78, 163.15, 78.65) mm, rotated rx 180 ry 0 rz -180 deg; joints [-145.777, -82.618, -27.406, 63.278, 39.025, -57.056]
  MoveL 5296 to (231.78, 163.15, 78.65) mm, rotated rx 180 ry 0 rz -180 deg; joints [-145.777, -82.618, -27.406, 63.278, 39.025, -57.056]
  Call Extruder(269.68807)
  MoveL 5297 to (231.54, 163.24, 78.65) mm, rotated rx 180 ry 0 rz 180 deg; joints [-145.759, -82.588, -27.468, 63.259, 39.055, -57.024]
  MoveL 5298 to (231.54, 163.24, 78.65) mm, rotated rx 180 ry 0 rz 180 deg; joints [-145.759, -82.588, -27.468, 63.259, 39.055, -57.024]
  Call Extruder(269.80129)
  MoveL 5299 to (231.35, 163.3, 78.65) mm, rotated rx 180 ry 0 rz -180 deg; joints [-145.744, -82.563, -27.519, 63.243, 39.078, -56.997]
  MoveL 5300 to (231.35, 163.3, 78.65) mm, rotated rx 180 ry 0 rz -180 deg; joints [-145.744, -82.563, -27.519, 63.243, 39.078, -56.997]
  Call Extruder(269.91407)
  MoveL 5301 to (231.17, 163.36, 78.65) mm, rotated rx -180 ry 0 rz 180 deg; joints [-145.73, -82.538, -27.569, 63.227, 39.102, -56.97]
  MoveL 5302 to (231.17, 163.36, 78.65) mm, rotated rx -180 ry 0 rz 180 deg; joints [-145.73, -82.538, -27.569, 63.227, 39.102, -56.97]
  Call Extruder(270.02640)
  MoveL 5303 to (230.98, 163.42, 78.65) mm, rotated rx -180 ry 0 rz 180 deg; joints [-145.716, -82.513, -27.62, 63.211, 39.125, -56.942]
  MoveL 5304 to (230.98, 163.42, 78.65) mm, rotated rx -180 ry 0 rz 180 deg; joints [-145.716, -82.513, -27.62, 63.211, 39.125, -56.942]
  Call Extruder(270.13829)
  MoveL 5305 to (230.79, 163.48, 78.65) mm, rotated rx 180 ry 0 rz -180 deg; joints [-145.702, -82.488, -27.671, 63.195, 39.149, -56.916]
  MoveL 5306 to (230.79, 163.48, 78.65) mm, rotated rx 180 ry 0 rz -180 deg; joints [-145.702, -82.488, -27.671, 63.195, 39.149, -56.916]
  Call Extruder(270.25969)
  MoveL 5307 to (230.58, 163.55, 78.65) mm, rotated rx -180 ry 0 rz 180 deg; joints [-145.687, -82.461, -27.726, 63.177, 39.174, -56.886]
  MoveL 5308 to (230.58, 163.55, 78.65) mm, rotated rx -180 ry 0 rz 180 deg; joints [-145.687, -82.461, -27.726, 63.177, 39.174, -56.886]
  Call Extruder(270.39051)
  MoveL 5309 to (230.36, 163.61, 78.65) mm, rotated rx 180 ry 0 rz 180 deg; joints [-145.67, -82.431, -27.787, 63.157, 39.202, -56.853]
  MoveL 5310 to (230.36, 163.61, 78.65) mm, rotated rx 180 ry 0 rz 180 deg; joints [-145.67, -82.431, -27.787, 63.157, 39.202, -56.853]
  Call Extruder(270.52075)
  MoveL 5311 to (230.14, 163.68, 78.65) mm, rotated rx 180 ry 0 rz 180 deg; joints [-145.654, -82.401, -27.848, 63.138, 39.23, -56.82]
  MoveL 5312 to (230.14, 163.68, 78.65) mm, rotated rx 180 ry 0 rz 180 deg; joints [-145.654, -82.401, -27.848, 63.138, 39.23, -56.82]
  Call Extruder(270.65044)
  MoveL 5313 to (229.91, 163.75, 78.65) mm, rotated rx 180 ry 0 rz 180 deg; joints [-145.638, -82.371, -27.909, 63.118, 39.257, -56.788]
  MoveL 5314 to (229.91, 163.75, 78.65) mm, rotated rx 180 ry 0 rz 180 deg; joints [-145.638, -82.371, -27.909, 63.118, 39.257, -56.788]
  Call Extruder(270.77955)
  MoveL 5315 to (229.69, 163.82, 78.65) mm, rotated rx 180 ry 0 rz -180 deg; joints [-145.621, -82.342, -27.97, 63.098, 39.285, -56.755]
  MoveL 5316 to (229.69, 163.82, 78.65) mm, rotated rx 180 ry 0 rz -180 deg; joints [-145.621, -82.342, -27.97, 63.098, 39.285, -56.755]
  Call Extruder(270.89463)
  MoveL 5317 to (229.48, 163.86, 78.65) mm, rotated rx 180 ry 0 rz 180 deg; joints [-145.607, -82.313, -28.029, 63.078, 39.31, -56.722]
  MoveL 5318 to (229.48, 163.86, 78.65) mm, rotated rx 180 ry 0 rz 180 deg; joints [-145.607, -82.313, -28.029, 63.078, 39.31, -56.722]
  Call Extruder(271.00925)
  MoveL 5319 to (229.28, 163.91, 78.65) mm, rotated rx 180 ry 0 rz -180 deg; joints [-145.594, -82.284, -28.088, 63.057, 39.335, -56.689]
  MoveL 5320 to (229.28, 163.91, 78.65) mm, rotated rx 180 ry 0 rz -180 deg; joints [-145.594, -82.284, -28.088, 63.057, 39.335, -56.689]
  Call Extruder(271.12342)
  MoveL 5321 to (229.08, 163.95, 78.65) mm, rotated rx -180 ry 0 rz -180 deg; joints [-145.58, -82.255, -28.147, 63.036, 39.361, -56.656]
  MoveL 5322 to (229.08, 163.95, 78.65) mm, rotated rx -180 ry 0 rz -180 deg; joints [-145.58, -82.255, -28.147, 63.036, 39.361, -56.656]
  Call Extruder(271.23713)
  MoveL 5323 to (228.87, 164, 78.65) mm, rotated rx -180 ry 0 rz 180 deg; joints [-145.566, -82.226, -28.206, 63.015, 39.386, -56.622]
  MoveL 5324 to (228.87, 164, 78.65) mm, rotated rx -180 ry 0 rz 180 deg; joints [-145.566, -82.226, -28.206, 63.015, 39.386, -56.622]
  Call Extruder(271.36255)
  MoveL 5325 to (228.65, 164.04, 78.65) mm, rotated rx 180 ry 0 rz 180 deg; joints [-145.551, -82.193, -28.272, 62.992, 39.413, -56.586]
